// TIA Portal project "Homework-Traffic Light" (V16)

(* hardware
DEVICE "HMI_1"  KTP700 Basic PN
   slot 0: "HMI_1"  KTP700 Basic PN  6AV2 123-2GB03-0AX0  16.0.0.0
   slot 1: "HMI_RT_1"  KTP700 Basic PN  6AV2 123-2GB03-0AX0  16.0.0.0
   slot 5: "HMI_1.IE_CP_1"  PROFINET Interface  16.0.0.0
      slot 1: "PROFINET Interface_1"  PROFINET Interface
         slot 1: "Port_1"  Port
DEVICE "PC-System_1"  SIMATIC PC station
   slot 0: "SIMATIC PC station"  Rail  SIMATIC PC-Station  V1.0
      slot 125: "Stationmanager"  Station_Manager  V6.0.4
   slot 1: "HMI_RT_2"  WinCC RT Advanced  6AV2 104-0xxxx-xxxx  16.0.0.0
      slot 33792: "Computer interface"  Host interface
   slot 2: "IE general_1"  IE General  IE_CP  V8.2.0
DEVICE "PC-System_2"  SIMATIC PC station
   slot 0: "SIMATIC PC station"  Rail  SIMATIC PC-Station  V1.0
      slot 125: "Stationmanager"  Station_Manager  V6.0.4
   slot 1: "HMI_RT_3"  WinCC RT Professional  6AV2 105-0xxxx-xxxx  16.0.0.0
   slot 2: "IE general_1"  IE General  IE_CP  V8.2.0
DEVICE "S71500/ET200MP station_1"  S7-1500 station
   slot 0: "Rail_0"  Rack  6ES7 590-1***0-0AA0
   slot 1: "PLC_2"  CPU 1512C-1 PN  6ES7 512-1CK00-0AB0  V2.5
      slot 3: "CPU display_1"  6ES7591-1AA00-0AA0
      slot 32768: "PROFINET interface_1"  X1
   slot 2: "CM PtP RS232 HF_1"  CM PtP RS232 HF  6ES7 541-1AD00-0AB0  V1.0
   slot 3: "CM PtP RS232 HF_2"  CM PtP RS232 HF  6ES7 541-1AD00-0AB0  V1.0
*)

// ===== PLC "PLC_2"  CPU 1512C-1 PN =====

VAR_GLOBAL   // PLC tag table "Default tag table"
   "System_Byte" AT %MB7 : Byte;
   "FirstScan" AT %M7.0 : Bool;
   "DiagStatusUpdate" AT %M7.1 : Bool;
   "AlwaysTRUE" AT %M7.2 : Bool;
   "AlwaysFALSE" AT %M7.3 : Bool;
   "Clock_Byte" AT %MB8 : Byte;
   "Clock_10Hz" AT %M8.0 : Bool;
   "Clock_5Hz" AT %M8.1 : Bool;
   "Clock_2.5Hz" AT %M8.2 : Bool;
   "Clock_2Hz" AT %M8.3 : Bool;
   "Clock_1.25Hz" AT %M8.4 : Bool;
   "Clock_1Hz" AT %M8.5 : Bool;
   "Clock_0.625Hz" AT %M8.6 : Bool;
   "Clock_0.5Hz" AT %M8.7 : Bool;
   "Pulse1" AT %M0.0 : Bool;
   "Pulse2" AT %M0.1 : Bool;
   "Pulse3" AT %M0.2 : Bool;
   "Pulse4" AT %M0.3 : Bool;
   "Pulse5" AT %M0.4 : Bool;
   "Pulse6" AT %M0.5 : Bool;
   "Pulse_1s" AT %M0.6 : Bool;
   "Pulse7" AT %M0.7 : Bool;
   "Remain3" AT %M1.0 : Bool;
   "Remain1" AT %M1.1 : Bool;
   "Remain2" AT %M1.2 : Bool;
   "Remain4" AT %M1.3 : Bool;
   "Green_A" AT %Q4.0 : Bool;
   "Yellow_A" AT %Q4.1 : Bool;
   "Red_A" AT %Q4.2 : Bool;
   "Green_B" AT %Q4.3 : Bool;
   "Yellow_B" AT %Q4.4 : Bool;
   "Red_B" AT %Q4.5 : Bool;
   "Stop_System(1)" AT %I10.0 : Bool;
   "Start_System" AT %I10.1 : Bool;
   "Cross_Over" AT %M5.0 : Bool;
END_VAR

DATA_BLOCK "System Data"   // DB1
{ S7_Optimized_Access := 'TRUE' }
VERSION : 0.1
   VAR
      "Green A" : Bool;
      "Green B" : Bool;
      "Yellow A" : Bool;
      "Yellow B" : Bool;
      "Red A" : Bool;
      "Red B" : Bool;
      HMI_Update : Bool;
      Enable_PP1 : Bool;
      Enalbe_PP2 : Bool;
      Enalbe_PP3 : Bool;
      Start : Bool;
      Stop : Bool;
      RUN_System : Bool;
      HMI_SET : Bool;
      "Green A _Value" : DInt;
      "Green B_Value" : DInt;
      "Yellow A_value" : DInt;
      "Yellow B_value" : DInt;
      Red_A_value : DInt;
      Red_B_Value : DInt;
      HMI_Green_A : DInt;
      HMI_Green_B : DInt;
      HMI_Yellow_A : DInt;
      HMI_Yellow_B : DInt;
      HMI_Red_A : DInt;
      HMI_Red_B : DInt;
      Reset : Bool;
      Last_signal : Bool;
      Read_Time : DTL;
      RET_Val : Word;
      Time_day : Bool;
      Time_night : Bool;
      Visible_1 : Bool;
      Visible_2 : Bool;
      Mode : DInt;
      Cross : Bool;
   END_VAR
BEGIN
END_DATA_BLOCK

DATA_BLOCK "7SEG_Convert1"   // DB6
{ S7_Optimized_Access := 'TRUE' }
VERSION : 0.1
// stored: InstanceOfName Convert_BCD_7SEG
"Convert_BCD_7SEG"
BEGIN
END_DATA_BLOCK

DATA_BLOCK "Data"   // DB8
{ S7_Optimized_Access := 'TRUE' }
VERSION : 0.1
   VAR
      HMI_Cancel : Bool;
      "Green A _Value" : DInt;
      "Green B_Value" : DInt;
      "1Timer_TImerA" : DInt;
      "1Timer_TimerB" : DInt;
      "4Timer_Timer" : DInt;
      Counter_Time : DInt;
      Time_Max_Counter : DInt;
      "Yellow A_Value" : DInt;
      "Yellow B_Value" : DInt;
      "Red A_Value" : DInt;
      "Red B_Value" : DInt;
      GY_Value_A : DInt;
      GY_Value_B : DInt;
      "1Timer_Remain_LightB" : DInt;
      "1Timer_Remain_LightA" : DInt;
      TIme_LIGHT_A : DInt;
      Time_LIGHT_B : DInt;
      Timer_Light_YellowB_Remain : DInt;
      Timer_Light_YellowA_Remain : DInt;
      Counter_remain_Light_A : DInt;
      Counter_remain_Light_B : DInt;
      DEC_DIV_A : Int;
      DEC_DIV_B : Int;
      DEC_MOD_A : Int;
      DEC_MOD_B : Int;
      Remain_DEC_A : Int;
      Remain_DEC_B : Int;
      "7SEG_DIV_A" : Byte;
      "7SEG_MOD_A" : Byte;
      "7SEG_DIV_B" : Byte;
      "7SEG_MOD_B" : Byte;
      Cross_Remain : DInt;
   END_VAR
BEGIN
END_DATA_BLOCK

DATA_BLOCK "7SEG_Convert2"   // DB9
{ S7_Optimized_Access := 'TRUE' }
VERSION : 0.1
// stored: InstanceOfName Convert_BCD_7SEG
"Convert_BCD_7SEG"
BEGIN
END_DATA_BLOCK

DATA_BLOCK "7SEG_Convert3"   // DB10
{ S7_Optimized_Access := 'TRUE' }
VERSION : 0.1
// stored: InstanceOfName Convert_BCD_7SEG
"Convert_BCD_7SEG"
BEGIN
END_DATA_BLOCK

DATA_BLOCK "7SEG_Convert4"   // DB11
{ S7_Optimized_Access := 'TRUE' }
VERSION : 0.1
// stored: InstanceOfName Convert_BCD_7SEG
"Convert_BCD_7SEG"
BEGIN
END_DATA_BLOCK

// folder: System blocks/Program resources

DATA_BLOCK "Timer1"   // DB2
{ S7_Optimized_Access := 'TRUE' }
AUTHOR : Simatic
FAMILY : IEC
NAME : IEC_TMR
VERSION : 1.0
// stored: InstanceOfName IEC_TIMER
"IEC_TIMER"
BEGIN
END_DATA_BLOCK

DATA_BLOCK "Timer2"   // DB3
{ S7_Optimized_Access := 'TRUE' }
AUTHOR : Simatic
FAMILY : IEC
NAME : IEC_TMR
VERSION : 1.0
// stored: InstanceOfName IEC_TIMER
"IEC_TIMER"
BEGIN
END_DATA_BLOCK

DATA_BLOCK "Timer3"   // DB4
{ S7_Optimized_Access := 'TRUE' }
AUTHOR : Simatic
FAMILY : IEC
NAME : IEC_TMR
VERSION : 1.0
// stored: InstanceOfName IEC_TIMER
"IEC_TIMER"
BEGIN
END_DATA_BLOCK

DATA_BLOCK "Timer4"   // DB5
{ S7_Optimized_Access := 'TRUE' }
AUTHOR : Simatic
FAMILY : IEC
NAME : IEC_TMR
VERSION : 1.0
// stored: InstanceOfName IEC_TIMER
"IEC_TIMER"
BEGIN
END_DATA_BLOCK

DATA_BLOCK "T1"   // DB7
{ S7_Optimized_Access := 'TRUE' }
AUTHOR : Simatic
FAMILY : IEC
NAME : IEC_TMR
VERSION : 1.0
// stored: InstanceOfName IEC_TIMER
"IEC_TIMER"
BEGIN
END_DATA_BLOCK

DATA_BLOCK "T2"   // DB13
{ S7_Optimized_Access := 'TRUE' }
AUTHOR : Simatic
FAMILY : IEC
NAME : IEC_TMR
VERSION : 1.0
// stored: InstanceOfName IEC_TIMER
"IEC_TIMER"
BEGIN
END_DATA_BLOCK

// folder: (top level)

FUNCTION_BLOCK "Convert_BCD_7SEG"   // FB1, SCL
{ S7_Optimized_Access := 'TRUE' }
VERSION : 0.1
   VAR_INPUT
      BCD_Val : Int;
   END_VAR
   VAR_OUTPUT
      "7SEG_Val" : Byte;
   END_VAR
   VAR_TEMP
      tmp : Byte;
   END_VAR
BEGIN
   #tmp := 0;
   IF #BCD_Val =0 THEN
       #tmp := 63;
   END_IF;
   IF #BCD_Val = 1 THEN
       #tmp := 6;
   END_IF;
   IF #BCD_Val = 2 THEN
       #tmp := 91;
   END_IF;
   IF #BCD_Val = 3 THEN
       #tmp := 79;
   END_IF;
   IF #BCD_Val = 4 THEN
       #tmp := 102;
   END_IF;
   IF #BCD_Val = 5 THEN
       #tmp := 109;
   END_IF;
   IF #BCD_Val = 6 THEN
       #tmp := 125;
   END_IF;
   IF #BCD_Val = 7 THEN
       #tmp := 7;
   END_IF;
   IF #BCD_Val = 8 THEN
       #tmp := 127;
   END_IF;
   IF #BCD_Val = 9 THEN
       #tmp := 111;
   END_IF;
   #"7SEG_Val" := #tmp;
END_FUNCTION_BLOCK

FUNCTION "PP2_4Timer" : Void   // FC1, LAD
{ S7_Optimized_Access := 'TRUE' }
VERSION : 0.1
   VAR_TEMP   // added for the SCL form of the ladder/FBD networks
      _w1 : Bool;
   END_VAR
BEGIN

REGION Network 1
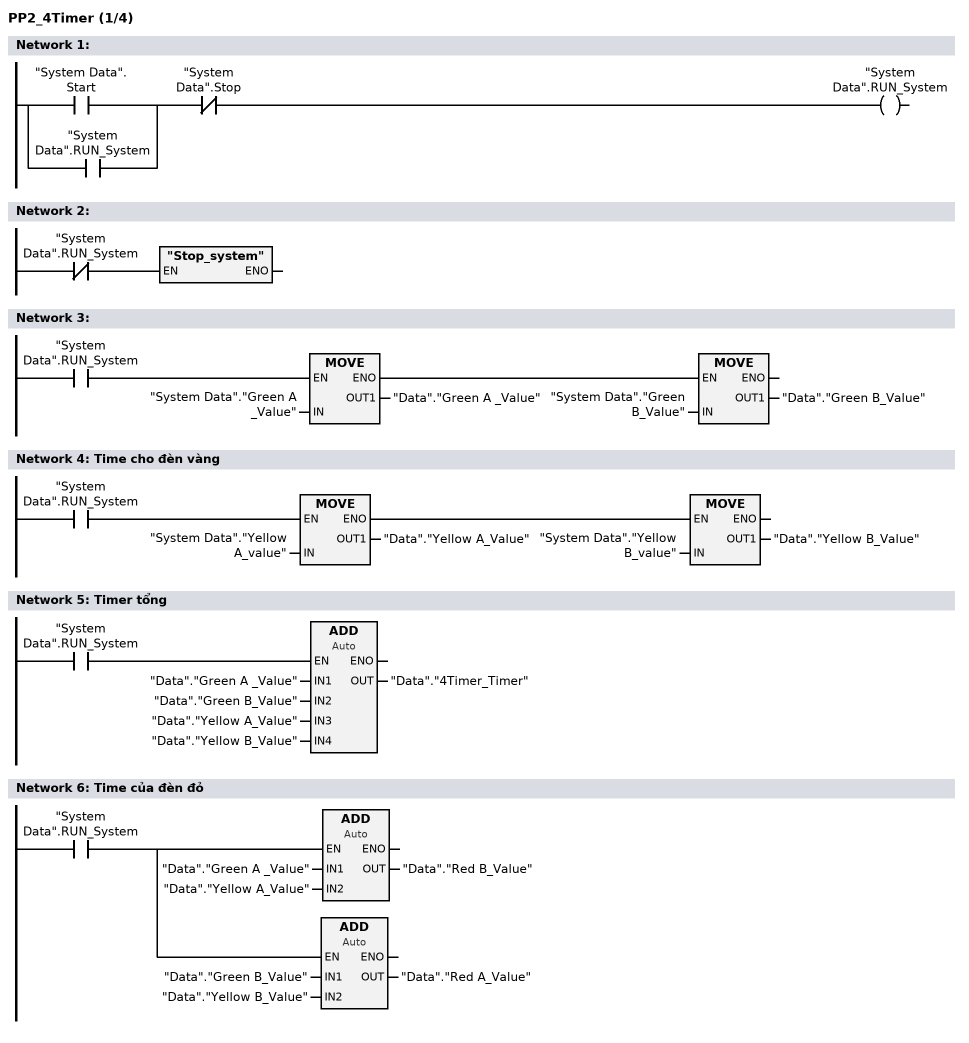
   RUNG wire#powerrail
      Contact( "System Data".Start )
      wire#w1
      I_Contact( "System Data".Stop )
      Coil( "System Data".RUN_System )
   END_RUNG
   RUNG wire#powerrail
      Contact( "System Data".RUN_System )
   END_RUNG wire#w1
   // the same network as SCL:
   "System Data".RUN_System := ("System Data".Start OR "System Data".RUN_System) AND NOT "System Data".Stop;
END_REGION

REGION Network 2
   RUNG wire#powerrail
      I_Contact( "System Data".RUN_System )
      "Stop_system"()
   END_RUNG
   // the same network as SCL:
   IF NOT "System Data".RUN_System THEN "Stop_system"(); END_IF;
END_REGION

REGION Network 3
   RUNG wire#powerrail
      Contact( "System Data".RUN_System )
      Move(in := "System Data"."Green A _Value", out1 => "Data"."Green A _Value")
      Move(in := "System Data"."Green B_Value", out1 => "Data"."Green B_Value")
   END_RUNG
   // the same network as SCL:
   IF "System Data".RUN_System THEN
       "Data"."Green A _Value" := "System Data"."Green A _Value";
       "Data"."Green B_Value" := "System Data"."Green B_Value";
   END_IF;
END_REGION

REGION Network 4: Time cho đèn vàng
   RUNG wire#powerrail
      Contact( "System Data".RUN_System )
      Move(in := "System Data"."Yellow A_value", out1 => "Data"."Yellow A_Value")
      Move(in := "System Data"."Yellow B_value", out1 => "Data"."Yellow B_Value")
   END_RUNG
   // the same network as SCL:
   IF "System Data".RUN_System THEN
       "Data"."Yellow A_Value" := "System Data"."Yellow A_value";
       "Data"."Yellow B_Value" := "System Data"."Yellow B_value";
   END_IF;
END_REGION

REGION Network 5: Timer tổng
   RUNG wire#powerrail
      Contact( "System Data".RUN_System )
      Add(in1 := "Data"."Green A _Value", in2 := "Data"."Green B_Value", in3 := "Data"."Yellow A_Value", in4 := "Data"."Yellow B_Value", out => "Data"."4Timer_Timer")
   END_RUNG
   // the same network as SCL:
   IF "System Data".RUN_System THEN
       "Data"."4Timer_Timer" := "Data"."Green A _Value" + "Data"."Green B_Value" + "Data"."Yellow A_Value" + "Data"."Yellow B_Value";
   END_IF;
END_REGION

REGION Network 6: Time của đèn đỏ
   RUNG wire#powerrail
      Contact( "System Data".RUN_System )
      wire#w1
      Add(in1 := "Data"."Green A _Value", in2 := "Data"."Yellow A_Value", out => "Data"."Red B_Value")
   END_RUNG
   RUNG wire#w1
      Add(in1 := "Data"."Green B_Value", in2 := "Data"."Yellow B_Value", out => "Data"."Red A_Value")
   END_RUNG
   // the same network as SCL:
   IF "System Data".RUN_System THEN
       "Data"."Red B_Value" := "Data"."Green A _Value" + "Data"."Yellow A_Value";
       "Data"."Red A_Value" := "Data"."Green B_Value" + "Data"."Yellow B_Value";
   END_IF;
END_REGION

REGION Network 7
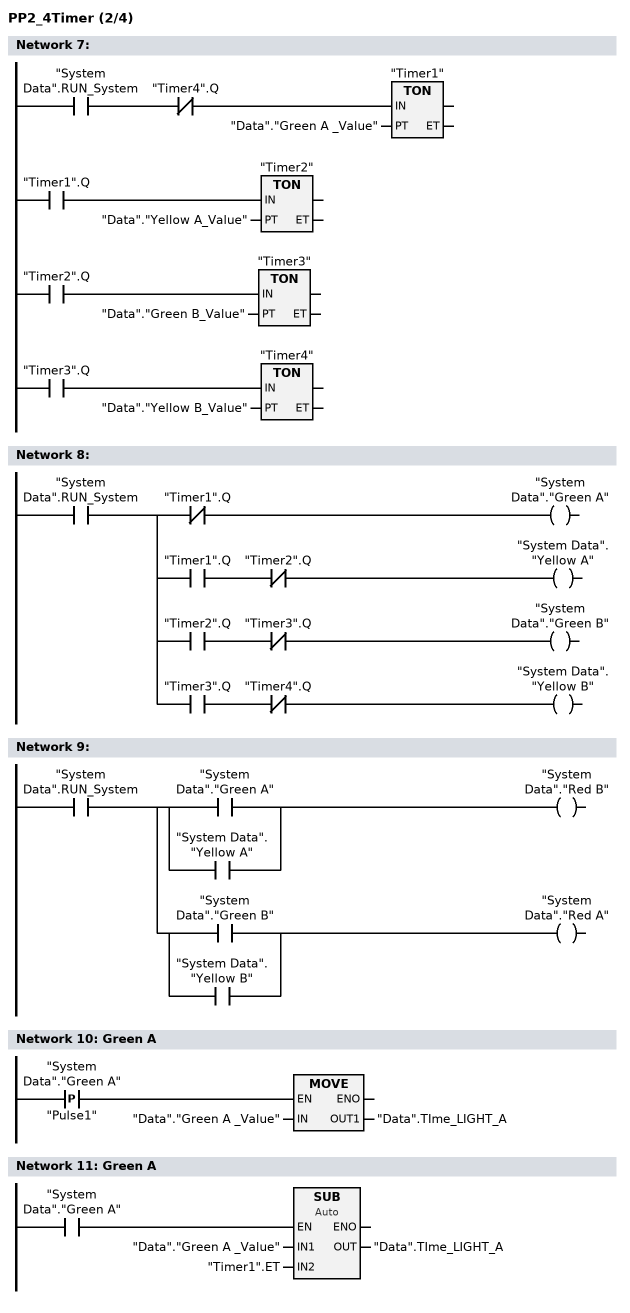
   "Timer1".TON(IN := "System Data".RUN_System AND NOT "Timer4".Q, PT := "Data"."Green A _Value");
   "Timer2".TON(IN := "Timer1".Q, PT := "Data"."Yellow A_Value");
   "Timer3".TON(IN := "Timer2".Q, PT := "Data"."Green B_Value");
   "Timer4".TON(IN := "Timer3".Q, PT := "Data"."Yellow B_Value");
END_REGION

REGION Network 8
   RUNG wire#powerrail
      Contact( "System Data".RUN_System )
      wire#w1
      I_Contact( "Timer1".Q )
      Coil( "System Data"."Green A" )
   END_RUNG
   RUNG wire#w1
      Contact( "Timer1".Q )
      I_Contact( "Timer2".Q )
      Coil( "System Data"."Yellow A" )
   END_RUNG
   RUNG wire#w1
      Contact( "Timer2".Q )
      I_Contact( "Timer3".Q )
      Coil( "System Data"."Green B" )
   END_RUNG
   RUNG wire#w1
      Contact( "Timer3".Q )
      I_Contact( "Timer4".Q )
      Coil( "System Data"."Yellow B" )
   END_RUNG
   // the same network as SCL:
   "System Data"."Green A" := "System Data".RUN_System AND NOT "Timer1".Q;
   "System Data"."Yellow A" := "System Data".RUN_System AND "Timer1".Q AND NOT "Timer2".Q;
   "System Data"."Green B" := "System Data".RUN_System AND "Timer2".Q AND NOT "Timer3".Q;
   "System Data"."Yellow B" := "System Data".RUN_System AND "Timer3".Q AND NOT "Timer4".Q;
END_REGION

REGION Network 9
   RUNG wire#powerrail
      Contact( "System Data".RUN_System )
      wire#w1
      Contact( "System Data"."Green A" )
      wire#w2
      Coil( "System Data"."Red B" )
   END_RUNG
   RUNG wire#w1
      Contact( "System Data"."Yellow A" )
   END_RUNG wire#w2
   RUNG wire#w1
      Contact( "System Data"."Green B" )
      wire#w3
      Coil( "System Data"."Red A" )
   END_RUNG
   RUNG wire#w1
      Contact( "System Data"."Yellow B" )
   END_RUNG wire#w3
   // the same network as SCL:
   "System Data"."Red B" := "System Data".RUN_System AND ("System Data"."Green A" OR "System Data"."Yellow A");
   "System Data"."Red A" := "System Data".RUN_System AND ("System Data"."Green B" OR "System Data"."Yellow B");
END_REGION

REGION Network 10: Green A
   RUNG wire#powerrail
      P_Contact(operand := "System Data"."Green A", bit := "Pulse1")
      Move(in := "Data"."Green A _Value", out1 => "Data".TIme_LIGHT_A)
   END_RUNG
   // the same network as SCL:
   #_w1 := "System Data"."Green A" AND NOT "Pulse1";   // rising edge of "System Data"."Green A"
   "Pulse1" := "System Data"."Green A";
   IF #_w1 THEN "Data".TIme_LIGHT_A := "Data"."Green A _Value"; END_IF;
END_REGION

REGION Network 11: Green A
   RUNG wire#powerrail
      Contact( "System Data"."Green A" )
      Sub(in1 := "Data"."Green A _Value", in2 := "Timer1".ET, out => "Data".TIme_LIGHT_A)
   END_RUNG
   // the same network as SCL:
   IF "System Data"."Green A" THEN "Data".TIme_LIGHT_A := "Data"."Green A _Value" - "Timer1".ET; END_IF;
END_REGION

REGION Network 12: Yellow A
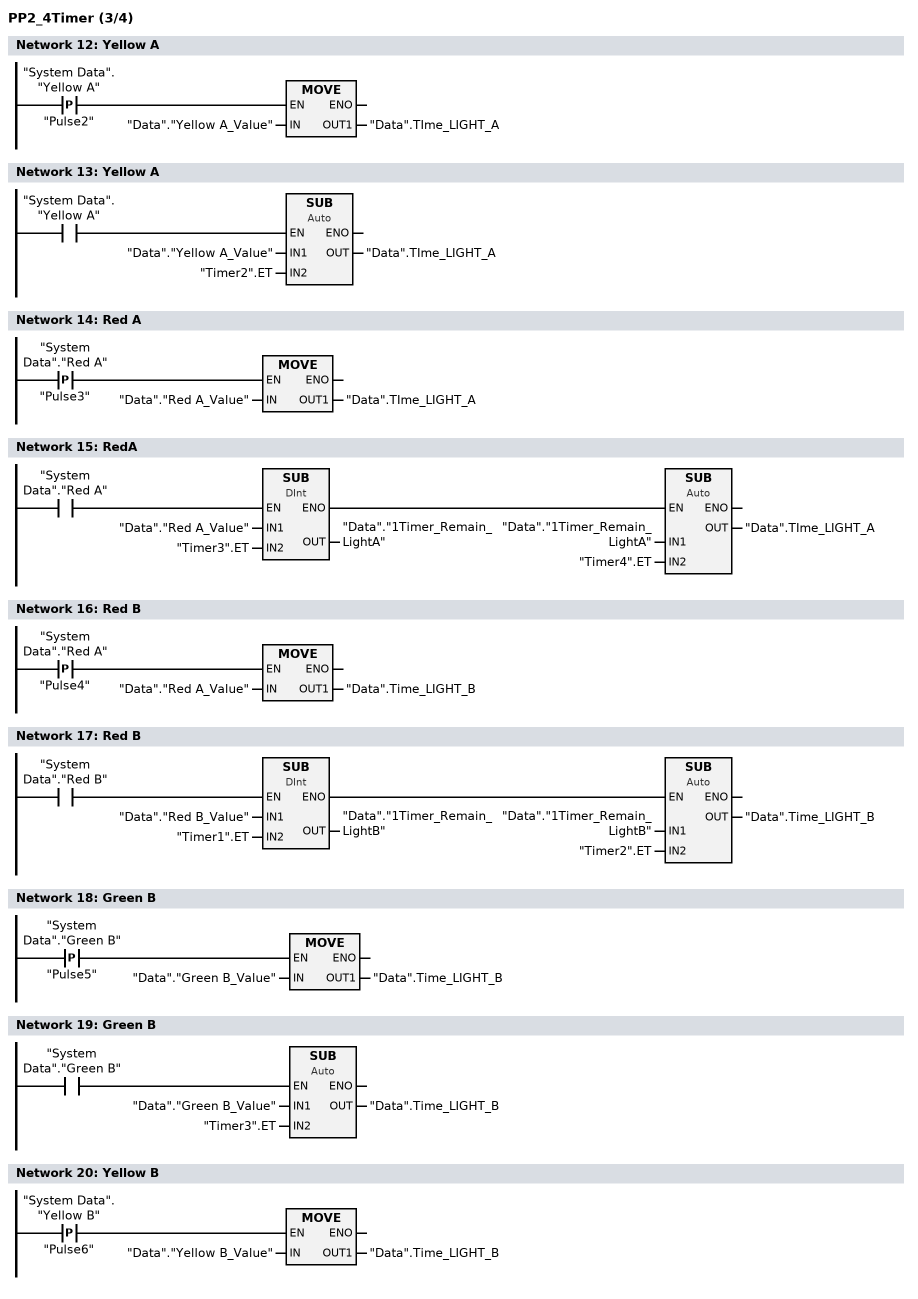
   RUNG wire#powerrail
      P_Contact(operand := "System Data"."Yellow A", bit := "Pulse2")
      Move(in := "Data"."Yellow A_Value", out1 => "Data".TIme_LIGHT_A)
   END_RUNG
   // the same network as SCL:
   #_w1 := "System Data"."Yellow A" AND NOT "Pulse2";   // rising edge of "System Data"."Yellow A"
   "Pulse2" := "System Data"."Yellow A";
   IF #_w1 THEN "Data".TIme_LIGHT_A := "Data"."Yellow A_Value"; END_IF;
END_REGION

REGION Network 13: Yellow A
   RUNG wire#powerrail
      Contact( "System Data"."Yellow A" )
      Sub(in1 := "Data"."Yellow A_Value", in2 := "Timer2".ET, out => "Data".TIme_LIGHT_A)
   END_RUNG
   // the same network as SCL:
   IF "System Data"."Yellow A" THEN "Data".TIme_LIGHT_A := "Data"."Yellow A_Value" - "Timer2".ET; END_IF;
END_REGION

REGION Network 14: Red A
   RUNG wire#powerrail
      P_Contact(operand := "System Data"."Red A", bit := "Pulse3")
      Move(in := "Data"."Red A_Value", out1 => "Data".TIme_LIGHT_A)
   END_RUNG
   // the same network as SCL:
   #_w1 := "System Data"."Red A" AND NOT "Pulse3";   // rising edge of "System Data"."Red A"
   "Pulse3" := "System Data"."Red A";
   IF #_w1 THEN "Data".TIme_LIGHT_A := "Data"."Red A_Value"; END_IF;
END_REGION

REGION Network 15: RedA
   RUNG wire#powerrail
      Contact( "System Data"."Red A" )
      { S7_Templates := "SrcType := DInt" } Sub(in1 := "Data"."Red A_Value", in2 := "Timer3".ET, out => "Data"."1Timer_Remain_LightA")
      Sub(in1 := "Data"."1Timer_Remain_LightA", in2 := "Timer4".ET, out => "Data".TIme_LIGHT_A)
   END_RUNG
   // the same network as SCL:
   IF "System Data"."Red A" THEN
       "Data"."1Timer_Remain_LightA" := "Data"."Red A_Value" - "Timer3".ET;
       "Data".TIme_LIGHT_A := "Data"."1Timer_Remain_LightA" - "Timer4".ET;
   END_IF;
END_REGION

REGION Network 16: Red B
   RUNG wire#powerrail
      P_Contact(operand := "System Data"."Red A", bit := "Pulse4")
      Move(in := "Data"."Red A_Value", out1 => "Data".Time_LIGHT_B)
   END_RUNG
   // the same network as SCL:
   #_w1 := "System Data"."Red A" AND NOT "Pulse4";   // rising edge of "System Data"."Red A"
   "Pulse4" := "System Data"."Red A";
   IF #_w1 THEN "Data".Time_LIGHT_B := "Data"."Red A_Value"; END_IF;
END_REGION

REGION Network 17: Red B
   RUNG wire#powerrail
      Contact( "System Data"."Red B" )
      { S7_Templates := "SrcType := DInt" } Sub(in1 := "Data"."Red B_Value", in2 := "Timer1".ET, out => "Data"."1Timer_Remain_LightB")
      Sub(in1 := "Data"."1Timer_Remain_LightB", in2 := "Timer2".ET, out => "Data".Time_LIGHT_B)
   END_RUNG
   // the same network as SCL:
   IF "System Data"."Red B" THEN
       "Data"."1Timer_Remain_LightB" := "Data"."Red B_Value" - "Timer1".ET;
       "Data".Time_LIGHT_B := "Data"."1Timer_Remain_LightB" - "Timer2".ET;
   END_IF;
END_REGION

REGION Network 18: Green B
   RUNG wire#powerrail
      P_Contact(operand := "System Data"."Green B", bit := "Pulse5")
      Move(in := "Data"."Green B_Value", out1 => "Data".Time_LIGHT_B)
   END_RUNG
   // the same network as SCL:
   #_w1 := "System Data"."Green B" AND NOT "Pulse5";   // rising edge of "System Data"."Green B"
   "Pulse5" := "System Data"."Green B";
   IF #_w1 THEN "Data".Time_LIGHT_B := "Data"."Green B_Value"; END_IF;
END_REGION

REGION Network 19: Green B
   RUNG wire#powerrail
      Contact( "System Data"."Green B" )
      Sub(in1 := "Data"."Green B_Value", in2 := "Timer3".ET, out => "Data".Time_LIGHT_B)
   END_RUNG
   // the same network as SCL:
   IF "System Data"."Green B" THEN "Data".Time_LIGHT_B := "Data"."Green B_Value" - "Timer3".ET; END_IF;
END_REGION

REGION Network 20: Yellow B
   RUNG wire#powerrail
      P_Contact(operand := "System Data"."Yellow B", bit := "Pulse6")
      Move(in := "Data"."Yellow B_Value", out1 => "Data".Time_LIGHT_B)
   END_RUNG
   // the same network as SCL:
   #_w1 := "System Data"."Yellow B" AND NOT "Pulse6";   // rising edge of "System Data"."Yellow B"
   "Pulse6" := "System Data"."Yellow B";
   IF #_w1 THEN "Data".Time_LIGHT_B := "Data"."Yellow B_Value"; END_IF;
END_REGION

REGION Network 21: Yellow B
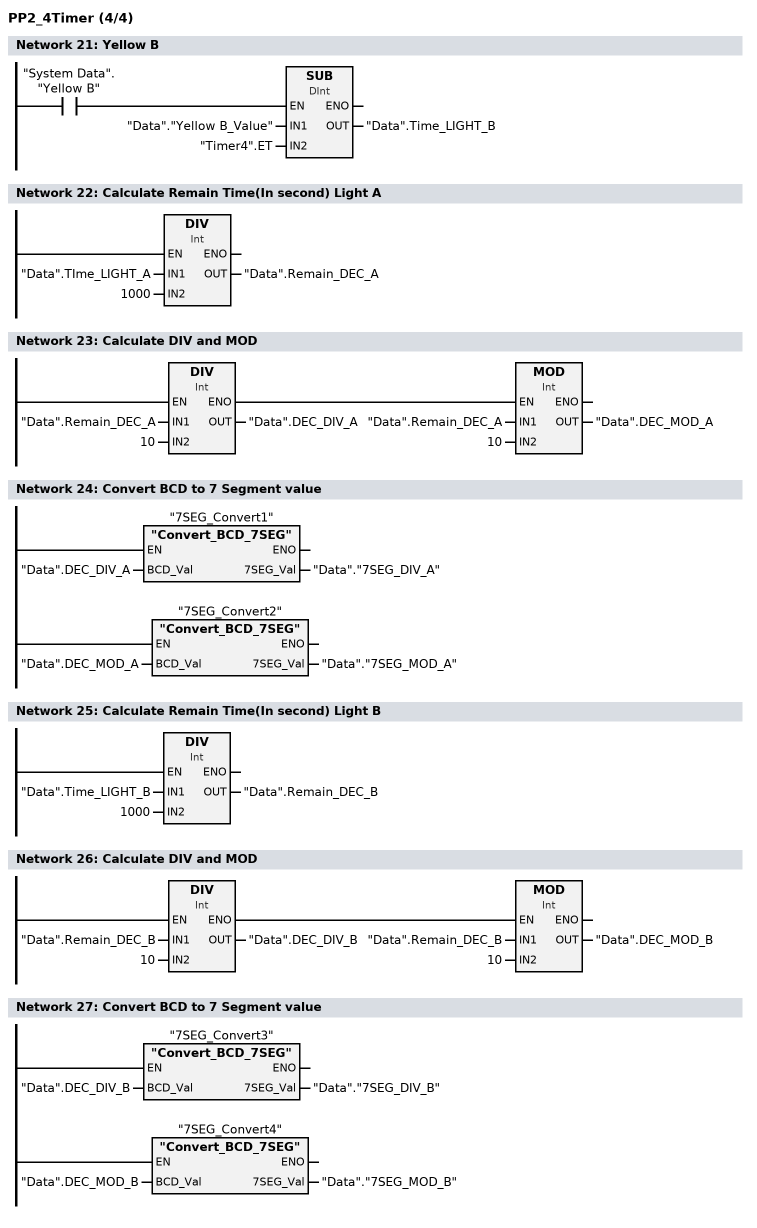
   RUNG wire#powerrail
      Contact( "System Data"."Yellow B" )
      { S7_Templates := "SrcType := DInt" } Sub(in1 := "Data"."Yellow B_Value", in2 := "Timer4".ET, out => "Data".Time_LIGHT_B)
   END_RUNG
   // the same network as SCL:
   IF "System Data"."Yellow B" THEN "Data".Time_LIGHT_B := "Data"."Yellow B_Value" - "Timer4".ET; END_IF;
END_REGION

REGION Network 22: Calculate Remain Time(In second) Light A
   RUNG wire#powerrail
      { S7_Templates := "SrcType := Int" } Div(in1 := "Data".TIme_LIGHT_A, in2 := 1000, out => "Data".Remain_DEC_A)
   END_RUNG
   // the same network as SCL:
   "Data".Remain_DEC_A := "Data".TIme_LIGHT_A / 1000;
END_REGION

REGION Network 23: Calculate DIV and MOD
   RUNG wire#powerrail
      { S7_Templates := "SrcType := Int" } Div(in1 := "Data".Remain_DEC_A, in2 := 10, out => "Data".DEC_DIV_A)
      { S7_Templates := "SrcType := Int" } Mod(in1 := "Data".Remain_DEC_A, in2 := 10, out => "Data".DEC_MOD_A)
   END_RUNG
   // the same network as SCL:
   "Data".DEC_DIV_A := "Data".Remain_DEC_A / 10;
   "Data".DEC_MOD_A := "Data".Remain_DEC_A MOD 10;
END_REGION

REGION Network 24: Convert BCD to 7 Segment value
   RUNG wire#powerrail
      "7SEG_Convert1"(BCD_Val := "Data".DEC_DIV_A, "7SEG_Val" => "Data"."7SEG_DIV_A")
   END_RUNG
   RUNG wire#powerrail
      "7SEG_Convert2"(BCD_Val := "Data".DEC_MOD_A, "7SEG_Val" => "Data"."7SEG_MOD_A")
   END_RUNG
   // the same network as SCL:
   "7SEG_Convert1"(BCD_Val := "Data".DEC_DIV_A, "7SEG_Val" => "Data"."7SEG_DIV_A");   // "Convert_BCD_7SEG"
   "7SEG_Convert2"(BCD_Val := "Data".DEC_MOD_A, "7SEG_Val" => "Data"."7SEG_MOD_A");   // "Convert_BCD_7SEG"
END_REGION

REGION Network 25: Calculate Remain Time(In second) Light B
   RUNG wire#powerrail
      { S7_Templates := "SrcType := Int" } Div(in1 := "Data".Time_LIGHT_B, in2 := 1000, out => "Data".Remain_DEC_B)
   END_RUNG
   // the same network as SCL:
   "Data".Remain_DEC_B := "Data".Time_LIGHT_B / 1000;
END_REGION

REGION Network 26: Calculate DIV and MOD
   RUNG wire#powerrail
      { S7_Templates := "SrcType := Int" } Div(in1 := "Data".Remain_DEC_B, in2 := 10, out => "Data".DEC_DIV_B)
      { S7_Templates := "SrcType := Int" } Mod(in1 := "Data".Remain_DEC_B, in2 := 10, out => "Data".DEC_MOD_B)
   END_RUNG
   // the same network as SCL:
   "Data".DEC_DIV_B := "Data".Remain_DEC_B / 10;
   "Data".DEC_MOD_B := "Data".Remain_DEC_B MOD 10;
END_REGION

REGION Network 27: Convert BCD to 7 Segment value
   RUNG wire#powerrail
      "7SEG_Convert3"(BCD_Val := "Data".DEC_DIV_B, "7SEG_Val" => "Data"."7SEG_DIV_B")
   END_RUNG
   RUNG wire#powerrail
      "7SEG_Convert4"(BCD_Val := "Data".DEC_MOD_B, "7SEG_Val" => "Data"."7SEG_MOD_B")
   END_RUNG
   // the same network as SCL:
   "7SEG_Convert3"(BCD_Val := "Data".DEC_DIV_B, "7SEG_Val" => "Data"."7SEG_DIV_B");   // "Convert_BCD_7SEG"
   "7SEG_Convert4"(BCD_Val := "Data".DEC_MOD_B, "7SEG_Val" => "Data"."7SEG_MOD_B");   // "Convert_BCD_7SEG"
END_REGION
END_FUNCTION

FUNCTION "PP1_1Timer" : Void   // FC2, LAD
{ S7_Optimized_Access := 'TRUE' }
VERSION : 0.1
   VAR_TEMP   // added for the SCL form of the ladder/FBD networks
      _w1 : Bool;
   END_VAR
BEGIN

REGION Network 1
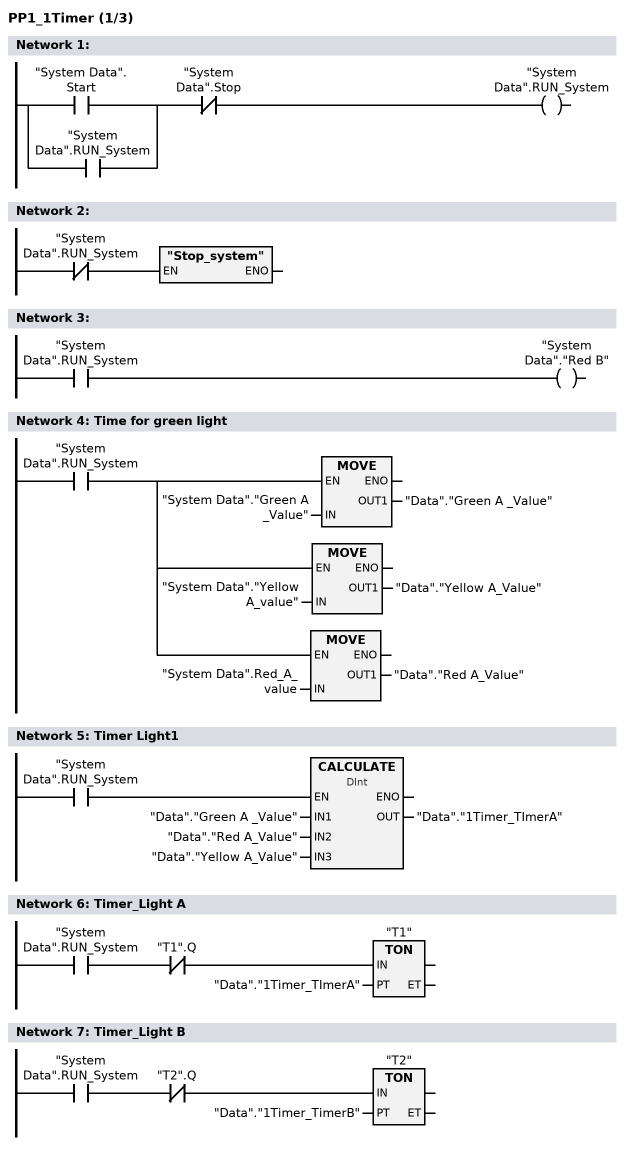
   RUNG wire#powerrail
      Contact( "System Data".Start )
      wire#w1
      I_Contact( "System Data".Stop )
      Coil( "System Data".RUN_System )
   END_RUNG
   RUNG wire#powerrail
      Contact( "System Data".RUN_System )
   END_RUNG wire#w1
   // the same network as SCL:
   "System Data".RUN_System := ("System Data".Start OR "System Data".RUN_System) AND NOT "System Data".Stop;
END_REGION

REGION Network 2
   RUNG wire#powerrail
      I_Contact( "System Data".RUN_System )
      "Stop_system"()
   END_RUNG
   // the same network as SCL:
   IF NOT "System Data".RUN_System THEN "Stop_system"(); END_IF;
END_REGION

REGION Network 3
   RUNG wire#powerrail
      Contact( "System Data".RUN_System )
      Coil( "System Data"."Red B" )
   END_RUNG
   // the same network as SCL:
   "System Data"."Red B" := "System Data".RUN_System;
END_REGION

REGION Network 4: Time for green light
   RUNG wire#powerrail
      Contact( "System Data".RUN_System )
      wire#w1
      Move(in := "System Data"."Green A _Value", out1 => "Data"."Green A _Value")
   END_RUNG
   RUNG wire#w1
      Move(in := "System Data"."Yellow A_value", out1 => "Data"."Yellow A_Value")
   END_RUNG
   RUNG wire#w1
      Move(in := "System Data".Red_A_value, out1 => "Data"."Red A_Value")
   END_RUNG
   // the same network as SCL:
   IF "System Data".RUN_System THEN
       "Data"."Green A _Value" := "System Data"."Green A _Value";
       "Data"."Yellow A_Value" := "System Data"."Yellow A_value";
       "Data"."Red A_Value" := "System Data".Red_A_value;
   END_IF;
END_REGION

REGION Network 5: Timer Light1
   RUNG wire#powerrail
      Contact( "System Data".RUN_System )
      { S7_Templates := "SrcType := DInt"; S7_Expression := "IN1+IN2+IN3" } Calculate(in1 := "Data"."Green A _Value", in2 := "Data"."Red A_Value", in3 := "Data"."Yellow A_Value", out => "Data"."1Timer_TImerA")
   END_RUNG
   // the same network as SCL:
   IF "System Data".RUN_System THEN
       "Data"."1Timer_TImerA" := "Data"."Green A _Value"+"Data"."Red A_Value"+"Data"."Yellow A_Value";
   END_IF;
END_REGION

REGION Network 6: Timer_Light A
   "T1".TON(IN := "System Data".RUN_System AND NOT "T1".Q, PT := "Data"."1Timer_TImerA");
END_REGION

REGION Network 7: Timer_Light B
   "T2".TON(IN := "System Data".RUN_System AND NOT "T2".Q, PT := "Data"."1Timer_TimerB");
END_REGION

REGION Network 8: Light A
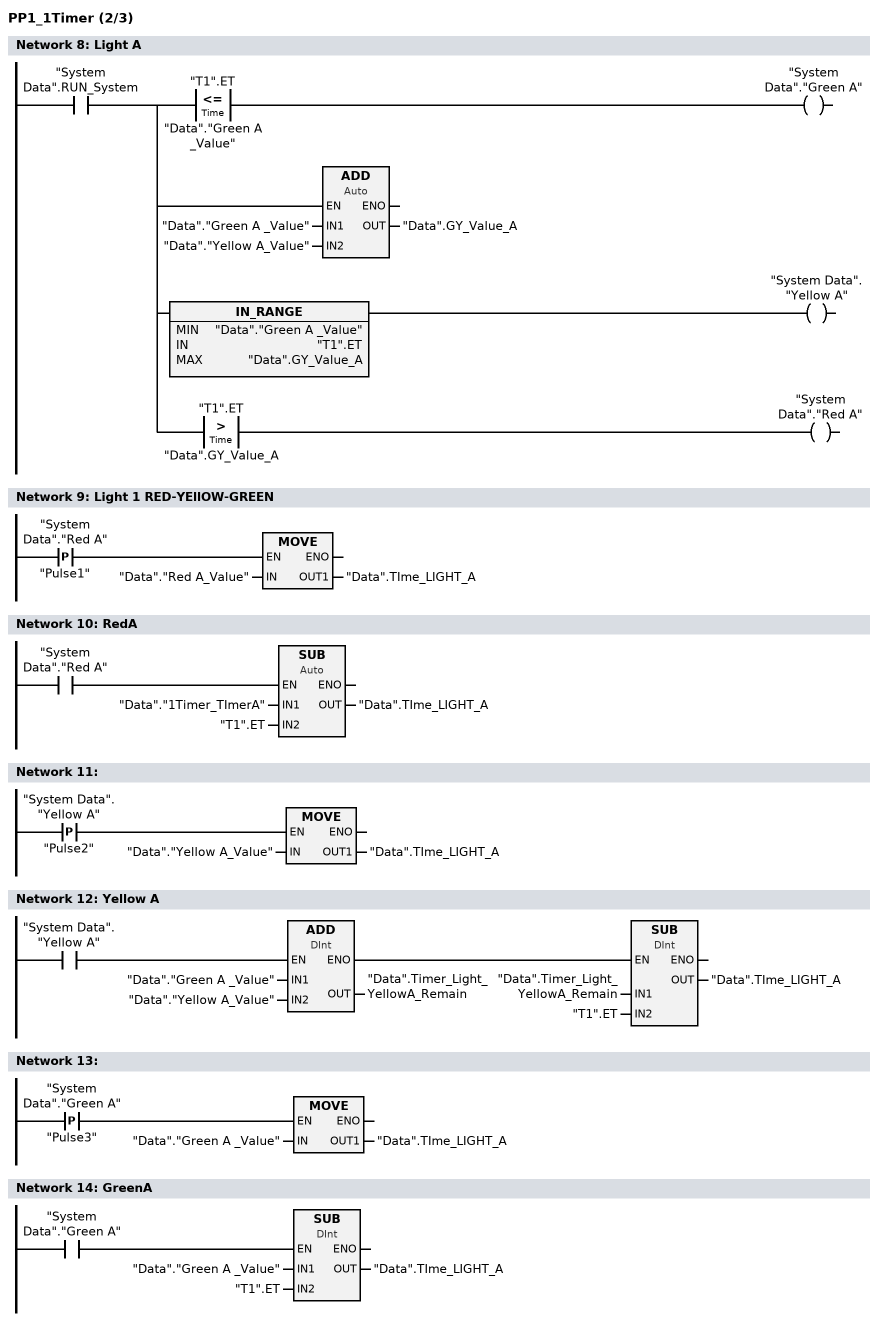
   RUNG wire#powerrail
      Contact( "System Data".RUN_System )
      wire#w1
      { S7_Templates := "SrcType := Time" } LE_Contact(in1 := "T1".ET, in2 := "Data"."Green A _Value")
      Coil( "System Data"."Green A" )
   END_RUNG
   RUNG wire#w1
      Add(in1 := "Data"."Green A _Value", in2 := "Data"."Yellow A_Value", out => "Data".GY_Value_A)
   END_RUNG
   RUNG wire#w1
      { S7_Templates := "SrcType := DInt" } InRange(min := "Data"."Green A _Value", in := "T1".ET, max := "Data".GY_Value_A)
      Coil( "System Data"."Yellow A" )
   END_RUNG
   RUNG wire#w1
      { S7_Templates := "SrcType := Time" } GT_Contact(in1 := "T1".ET, in2 := "Data".GY_Value_A)
      Coil( "System Data"."Red A" )
   END_RUNG
   // the same network as SCL:
   "System Data"."Green A" := "System Data".RUN_System AND ("T1".ET <= "Data"."Green A _Value");
   IF "System Data".RUN_System THEN
       "Data".GY_Value_A := "Data"."Green A _Value" + "Data"."Yellow A_Value";
   END_IF;
   "System Data"."Yellow A" := "System Data".RUN_System AND ("Data"."Green A _Value" <= "T1".ET) AND ("T1".ET <= "Data".GY_Value_A);
   "System Data"."Red A" := "System Data".RUN_System AND ("T1".ET > "Data".GY_Value_A);
END_REGION

REGION Network 9: Light 1 RED-YEllOW-GREEN
   RUNG wire#powerrail
      P_Contact(operand := "System Data"."Red A", bit := "Pulse1")
      Move(in := "Data"."Red A_Value", out1 => "Data".TIme_LIGHT_A)
   END_RUNG
   // the same network as SCL:
   #_w1 := "System Data"."Red A" AND NOT "Pulse1";   // rising edge of "System Data"."Red A"
   "Pulse1" := "System Data"."Red A";
   IF #_w1 THEN "Data".TIme_LIGHT_A := "Data"."Red A_Value"; END_IF;
END_REGION

REGION Network 10: RedA
   RUNG wire#powerrail
      Contact( "System Data"."Red A" )
      Sub(in1 := "Data"."1Timer_TImerA", in2 := "T1".ET, out => "Data".TIme_LIGHT_A)
   END_RUNG
   // the same network as SCL:
   IF "System Data"."Red A" THEN "Data".TIme_LIGHT_A := "Data"."1Timer_TImerA" - "T1".ET; END_IF;
END_REGION

REGION Network 11
   RUNG wire#powerrail
      P_Contact(operand := "System Data"."Yellow A", bit := "Pulse2")
      Move(in := "Data"."Yellow A_Value", out1 => "Data".TIme_LIGHT_A)
   END_RUNG
   // the same network as SCL:
   #_w1 := "System Data"."Yellow A" AND NOT "Pulse2";   // rising edge of "System Data"."Yellow A"
   "Pulse2" := "System Data"."Yellow A";
   IF #_w1 THEN "Data".TIme_LIGHT_A := "Data"."Yellow A_Value"; END_IF;
END_REGION

REGION Network 12: Yellow A
   RUNG wire#powerrail
      Contact( "System Data"."Yellow A" )
      { S7_Templates := "SrcType := DInt" } Add(in1 := "Data"."Green A _Value", in2 := "Data"."Yellow A_Value", out => "Data".Timer_Light_YellowA_Remain)
      { S7_Templates := "SrcType := DInt" } Sub(in1 := "Data".Timer_Light_YellowA_Remain, in2 := "T1".ET, out => "Data".TIme_LIGHT_A)
   END_RUNG
   // the same network as SCL:
   IF "System Data"."Yellow A" THEN
       "Data".Timer_Light_YellowA_Remain := "Data"."Green A _Value" + "Data"."Yellow A_Value";
       "Data".TIme_LIGHT_A := "Data".Timer_Light_YellowA_Remain - "T1".ET;
   END_IF;
END_REGION

REGION Network 13
   RUNG wire#powerrail
      P_Contact(operand := "System Data"."Green A", bit := "Pulse3")
      Move(in := "Data"."Green A _Value", out1 => "Data".TIme_LIGHT_A)
   END_RUNG
   // the same network as SCL:
   #_w1 := "System Data"."Green A" AND NOT "Pulse3";   // rising edge of "System Data"."Green A"
   "Pulse3" := "System Data"."Green A";
   IF #_w1 THEN "Data".TIme_LIGHT_A := "Data"."Green A _Value"; END_IF;
END_REGION

REGION Network 14: GreenA
   RUNG wire#powerrail
      Contact( "System Data"."Green A" )
      { S7_Templates := "SrcType := DInt" } Sub(in1 := "Data"."Green A _Value", in2 := "T1".ET, out => "Data".TIme_LIGHT_A)
   END_RUNG
   // the same network as SCL:
   IF "System Data"."Green A" THEN "Data".TIme_LIGHT_A := "Data"."Green A _Value" - "T1".ET; END_IF;
END_REGION

REGION Network 15: Calculate Remain Time(In second) Light A
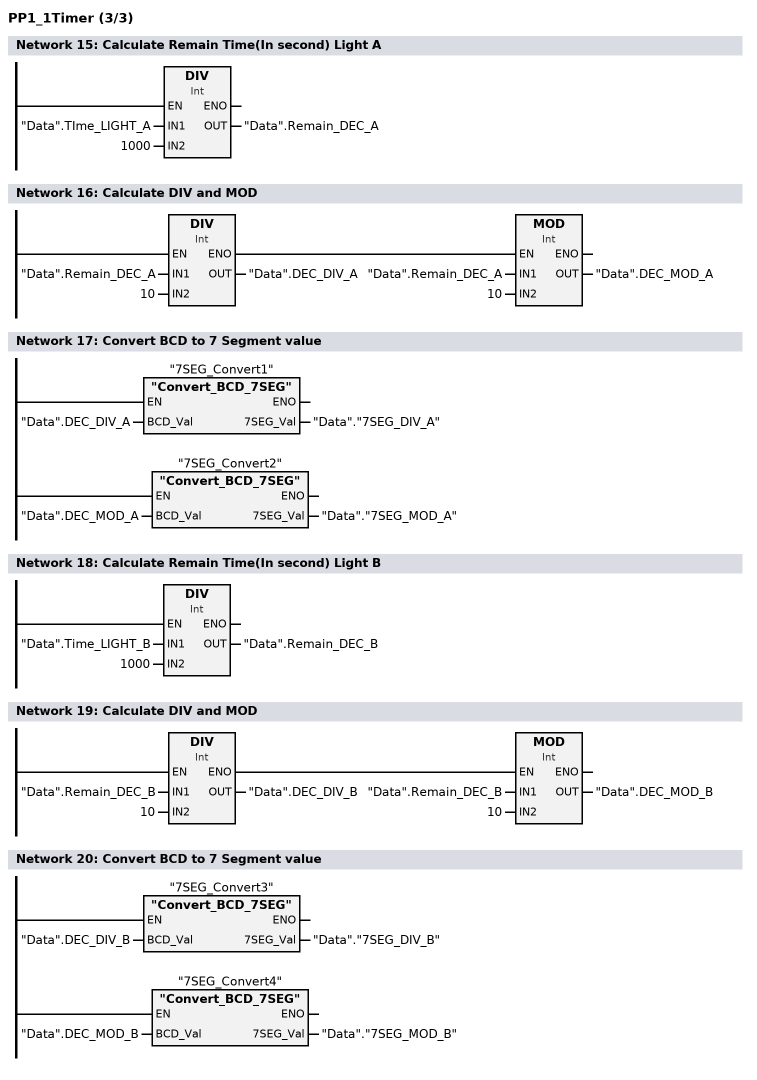
   RUNG wire#powerrail
      { S7_Templates := "SrcType := Int" } Div(in1 := "Data".TIme_LIGHT_A, in2 := 1000, out => "Data".Remain_DEC_A)
   END_RUNG
   // the same network as SCL:
   "Data".Remain_DEC_A := "Data".TIme_LIGHT_A / 1000;
END_REGION

REGION Network 16: Calculate DIV and MOD
   RUNG wire#powerrail
      { S7_Templates := "SrcType := Int" } Div(in1 := "Data".Remain_DEC_A, in2 := 10, out => "Data".DEC_DIV_A)
      { S7_Templates := "SrcType := Int" } Mod(in1 := "Data".Remain_DEC_A, in2 := 10, out => "Data".DEC_MOD_A)
   END_RUNG
   // the same network as SCL:
   "Data".DEC_DIV_A := "Data".Remain_DEC_A / 10;
   "Data".DEC_MOD_A := "Data".Remain_DEC_A MOD 10;
END_REGION

REGION Network 17: Convert BCD to 7 Segment value
   RUNG wire#powerrail
      "7SEG_Convert1"(BCD_Val := "Data".DEC_DIV_A, "7SEG_Val" => "Data"."7SEG_DIV_A")
   END_RUNG
   RUNG wire#powerrail
      "7SEG_Convert2"(BCD_Val := "Data".DEC_MOD_A, "7SEG_Val" => "Data"."7SEG_MOD_A")
   END_RUNG
   // the same network as SCL:
   "7SEG_Convert1"(BCD_Val := "Data".DEC_DIV_A, "7SEG_Val" => "Data"."7SEG_DIV_A");   // "Convert_BCD_7SEG"
   "7SEG_Convert2"(BCD_Val := "Data".DEC_MOD_A, "7SEG_Val" => "Data"."7SEG_MOD_A");   // "Convert_BCD_7SEG"
END_REGION

REGION Network 18: Calculate Remain Time(In second) Light B
   RUNG wire#powerrail
      { S7_Templates := "SrcType := Int" } Div(in1 := "Data".Time_LIGHT_B, in2 := 1000, out => "Data".Remain_DEC_B)
   END_RUNG
   // the same network as SCL:
   "Data".Remain_DEC_B := "Data".Time_LIGHT_B / 1000;
END_REGION

REGION Network 19: Calculate DIV and MOD
   RUNG wire#powerrail
      { S7_Templates := "SrcType := Int" } Div(in1 := "Data".Remain_DEC_B, in2 := 10, out => "Data".DEC_DIV_B)
      { S7_Templates := "SrcType := Int" } Mod(in1 := "Data".Remain_DEC_B, in2 := 10, out => "Data".DEC_MOD_B)
   END_RUNG
   // the same network as SCL:
   "Data".DEC_DIV_B := "Data".Remain_DEC_B / 10;
   "Data".DEC_MOD_B := "Data".Remain_DEC_B MOD 10;
END_REGION

REGION Network 20: Convert BCD to 7 Segment value
   RUNG wire#powerrail
      "7SEG_Convert3"(BCD_Val := "Data".DEC_DIV_B, "7SEG_Val" => "Data"."7SEG_DIV_B")
   END_RUNG
   RUNG wire#powerrail
      "7SEG_Convert4"(BCD_Val := "Data".DEC_MOD_B, "7SEG_Val" => "Data"."7SEG_MOD_B")
   END_RUNG
   // the same network as SCL:
   "7SEG_Convert3"(BCD_Val := "Data".DEC_DIV_B, "7SEG_Val" => "Data"."7SEG_DIV_B");   // "Convert_BCD_7SEG"
   "7SEG_Convert4"(BCD_Val := "Data".DEC_MOD_B, "7SEG_Val" => "Data"."7SEG_MOD_B");   // "Convert_BCD_7SEG"
END_REGION
END_FUNCTION

FUNCTION "PP3_Counter" : Void   // FC3, LAD
{ S7_Optimized_Access := 'TRUE' }
VERSION : 0.1
   VAR_TEMP   // added for the SCL form of the ladder/FBD networks
      _w1 : Bool;
   END_VAR
BEGIN

REGION Network 1: System
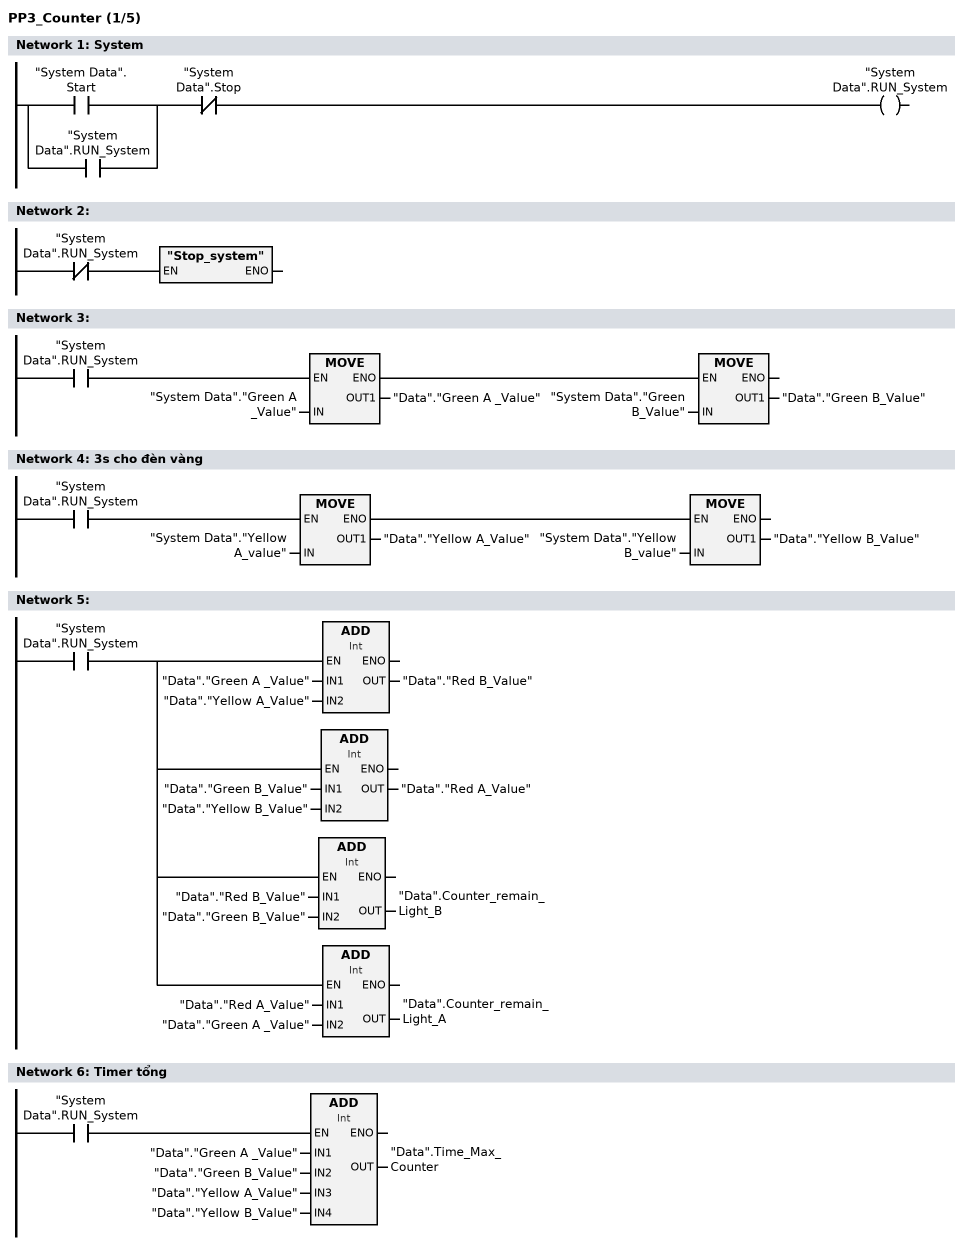
   RUNG wire#powerrail
      Contact( "System Data".Start )
      wire#w1
      I_Contact( "System Data".Stop )
      Coil( "System Data".RUN_System )
   END_RUNG
   RUNG wire#powerrail
      Contact( "System Data".RUN_System )
   END_RUNG wire#w1
   // the same network as SCL:
   "System Data".RUN_System := ("System Data".Start OR "System Data".RUN_System) AND NOT "System Data".Stop;
END_REGION

REGION Network 2
   RUNG wire#powerrail
      I_Contact( "System Data".RUN_System )
      "Stop_system"()
   END_RUNG
   // the same network as SCL:
   IF NOT "System Data".RUN_System THEN "Stop_system"(); END_IF;
END_REGION

REGION Network 3
   RUNG wire#powerrail
      Contact( "System Data".RUN_System )
      Move(in := "System Data"."Green A _Value", out1 => "Data"."Green A _Value")
      Move(in := "System Data"."Green B_Value", out1 => "Data"."Green B_Value")
   END_RUNG
   // the same network as SCL:
   IF "System Data".RUN_System THEN
       "Data"."Green A _Value" := "System Data"."Green A _Value";
       "Data"."Green B_Value" := "System Data"."Green B_Value";
   END_IF;
END_REGION

REGION Network 4: 3s cho đèn vàng
   RUNG wire#powerrail
      Contact( "System Data".RUN_System )
      Move(in := "System Data"."Yellow A_value", out1 => "Data"."Yellow A_Value")
      Move(in := "System Data"."Yellow B_value", out1 => "Data"."Yellow B_Value")
   END_RUNG
   // the same network as SCL:
   IF "System Data".RUN_System THEN
       "Data"."Yellow A_Value" := "System Data"."Yellow A_value";
       "Data"."Yellow B_Value" := "System Data"."Yellow B_value";
   END_IF;
END_REGION

REGION Network 5
   RUNG wire#powerrail
      Contact( "System Data".RUN_System )
      wire#w1
      { S7_Templates := "SrcType := Int" } Add(in1 := "Data"."Green A _Value", in2 := "Data"."Yellow A_Value", out => "Data"."Red B_Value")
   END_RUNG
   RUNG wire#w1
      { S7_Templates := "SrcType := Int" } Add(in1 := "Data"."Green B_Value", in2 := "Data"."Yellow B_Value", out => "Data"."Red A_Value")
   END_RUNG
   RUNG wire#w1
      { S7_Templates := "SrcType := Int" } Add(in1 := "Data"."Red B_Value", in2 := "Data"."Green B_Value", out => "Data".Counter_remain_Light_B)
   END_RUNG
   RUNG wire#w1
      { S7_Templates := "SrcType := Int" } Add(in1 := "Data"."Red A_Value", in2 := "Data"."Green A _Value", out => "Data".Counter_remain_Light_A)
   END_RUNG
   // the same network as SCL:
   IF "System Data".RUN_System THEN
       "Data"."Red B_Value" := "Data"."Green A _Value" + "Data"."Yellow A_Value";
       "Data"."Red A_Value" := "Data"."Green B_Value" + "Data"."Yellow B_Value";
       "Data".Counter_remain_Light_B := "Data"."Red B_Value" + "Data"."Green B_Value";
       "Data".Counter_remain_Light_A := "Data"."Red A_Value" + "Data"."Green A _Value";
   END_IF;
END_REGION

REGION Network 6: Timer tổng
   RUNG wire#powerrail
      Contact( "System Data".RUN_System )
      { S7_Templates := "SrcType := Int" } Add(in1 := "Data"."Green A _Value", in2 := "Data"."Green B_Value", in3 := "Data"."Yellow A_Value", in4 := "Data"."Yellow B_Value", out => "Data".Time_Max_Counter)
   END_RUNG
   // the same network as SCL:
   IF "System Data".RUN_System THEN
       "Data".Time_Max_Counter := "Data"."Green A _Value" + "Data"."Green B_Value" + "Data"."Yellow A_Value" + "Data"."Yellow B_Value";
   END_IF;
END_REGION

REGION Network 7: Tạo xung 1s
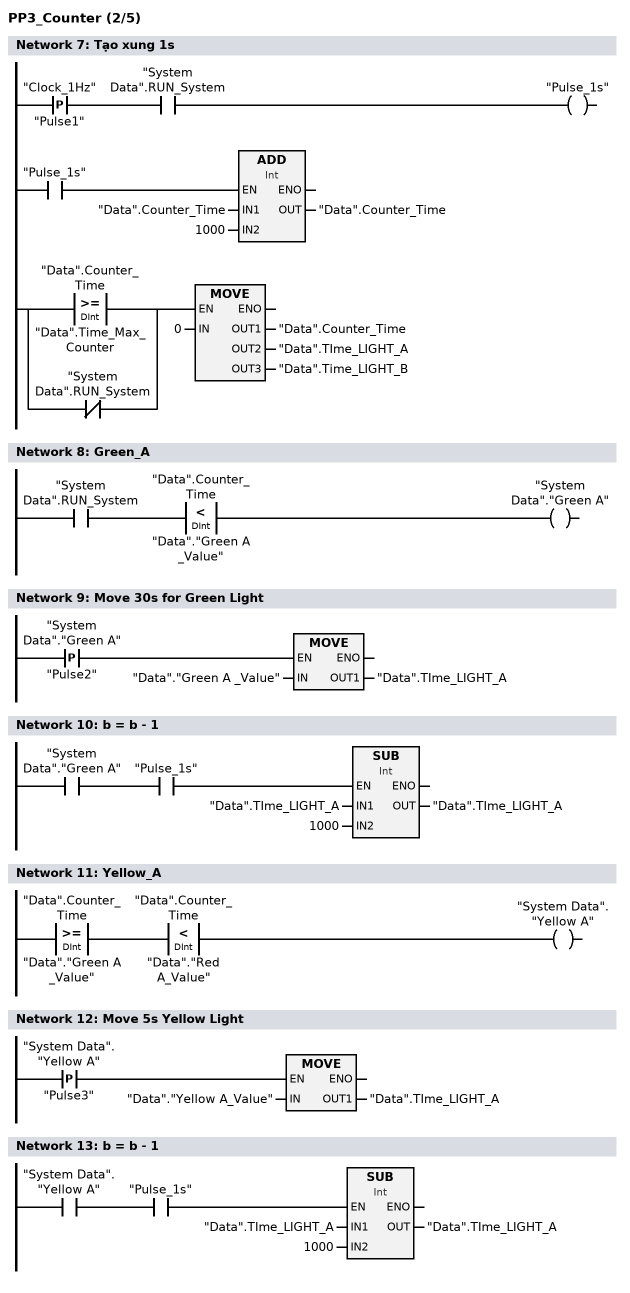
   RUNG wire#powerrail
      P_Contact(operand := "Clock_1Hz", bit := "Pulse1")
      Contact( "System Data".RUN_System )
      Coil( "Pulse_1s" )
   END_RUNG
   RUNG wire#powerrail
      Contact( "Pulse_1s" )
      { S7_Templates := "SrcType := Int" } Add(in1 := "Data".Counter_Time, in2 := 1000, out => "Data".Counter_Time)
   END_RUNG
   RUNG wire#powerrail
      { S7_Templates := "SrcType := DInt" } GE_Contact(in1 := "Data".Counter_Time, in2 := "Data".Time_Max_Counter)
      wire#w1
      Move(in := 0, out1 => "Data".Counter_Time, out2 => "Data".TIme_LIGHT_A, out3 => "Data".Time_LIGHT_B)
   END_RUNG
   RUNG wire#powerrail
      I_Contact( "System Data".RUN_System )
   END_RUNG wire#w1
   // the same network as SCL:
   #_w1 := "Clock_1Hz" AND NOT "Pulse1";   // rising edge of "Clock_1Hz"
   "Pulse1" := "Clock_1Hz";
   "Pulse_1s" := #_w1 AND "System Data".RUN_System;
   IF "Pulse_1s" THEN "Data".Counter_Time := "Data".Counter_Time + 1000; END_IF;
   IF ("Data".Counter_Time >= "Data".Time_Max_Counter) OR NOT "System Data".RUN_System THEN
       "Data".Counter_Time := 0;
       "Data".TIme_LIGHT_A := 0;
       "Data".Time_LIGHT_B := 0;
   END_IF;
END_REGION

REGION Network 8: Green_A
   RUNG wire#powerrail
      Contact( "System Data".RUN_System )
      { S7_Templates := "SrcType := DInt" } LT_Contact(in1 := "Data".Counter_Time, in2 := "Data"."Green A _Value")
      Coil( "System Data"."Green A" )
   END_RUNG
   // the same network as SCL:
   "System Data"."Green A" := "System Data".RUN_System AND ("Data".Counter_Time < "Data"."Green A _Value");
END_REGION

REGION Network 9: Move 30s for Green Light
   RUNG wire#powerrail
      P_Contact(operand := "System Data"."Green A", bit := "Pulse2")
      Move(in := "Data"."Green A _Value", out1 => "Data".TIme_LIGHT_A)
   END_RUNG
   // the same network as SCL:
   #_w1 := "System Data"."Green A" AND NOT "Pulse2";   // rising edge of "System Data"."Green A"
   "Pulse2" := "System Data"."Green A";
   IF #_w1 THEN "Data".TIme_LIGHT_A := "Data"."Green A _Value"; END_IF;
END_REGION

REGION Network 10: b = b - 1
   RUNG wire#powerrail
      Contact( "System Data"."Green A" )
      Contact( "Pulse_1s" )
      { S7_Templates := "SrcType := Int" } Sub(in1 := "Data".TIme_LIGHT_A, in2 := 1000, out => "Data".TIme_LIGHT_A)
   END_RUNG
   // the same network as SCL:
   IF "System Data"."Green A" AND "Pulse_1s" THEN "Data".TIme_LIGHT_A := "Data".TIme_LIGHT_A - 1000; END_IF;
END_REGION

REGION Network 11: Yellow_A
   RUNG wire#powerrail
      { S7_Templates := "SrcType := DInt" } GE_Contact(in1 := "Data".Counter_Time, in2 := "Data"."Green A _Value")
      { S7_Templates := "SrcType := DInt" } LT_Contact(in1 := "Data".Counter_Time, in2 := "Data"."Red A_Value")
      Coil( "System Data"."Yellow A" )
   END_RUNG
   // the same network as SCL:
   "System Data"."Yellow A" := ("Data".Counter_Time >= "Data"."Green A _Value") AND ("Data".Counter_Time < "Data"."Red A_Value");
END_REGION

REGION Network 12: Move 5s Yellow Light
   RUNG wire#powerrail
      P_Contact(operand := "System Data"."Yellow A", bit := "Pulse3")
      Move(in := "Data"."Yellow A_Value", out1 => "Data".TIme_LIGHT_A)
   END_RUNG
   // the same network as SCL:
   #_w1 := "System Data"."Yellow A" AND NOT "Pulse3";   // rising edge of "System Data"."Yellow A"
   "Pulse3" := "System Data"."Yellow A";
   IF #_w1 THEN "Data".TIme_LIGHT_A := "Data"."Yellow A_Value"; END_IF;
END_REGION

REGION Network 13: b = b - 1
   RUNG wire#powerrail
      Contact( "System Data"."Yellow A" )
      Contact( "Pulse_1s" )
      { S7_Templates := "SrcType := Int" } Sub(in1 := "Data".TIme_LIGHT_A, in2 := 1000, out => "Data".TIme_LIGHT_A)
   END_RUNG
   // the same network as SCL:
   IF "System Data"."Yellow A" AND "Pulse_1s" THEN "Data".TIme_LIGHT_A := "Data".TIme_LIGHT_A - 1000; END_IF;
END_REGION

REGION Network 14: Red_A
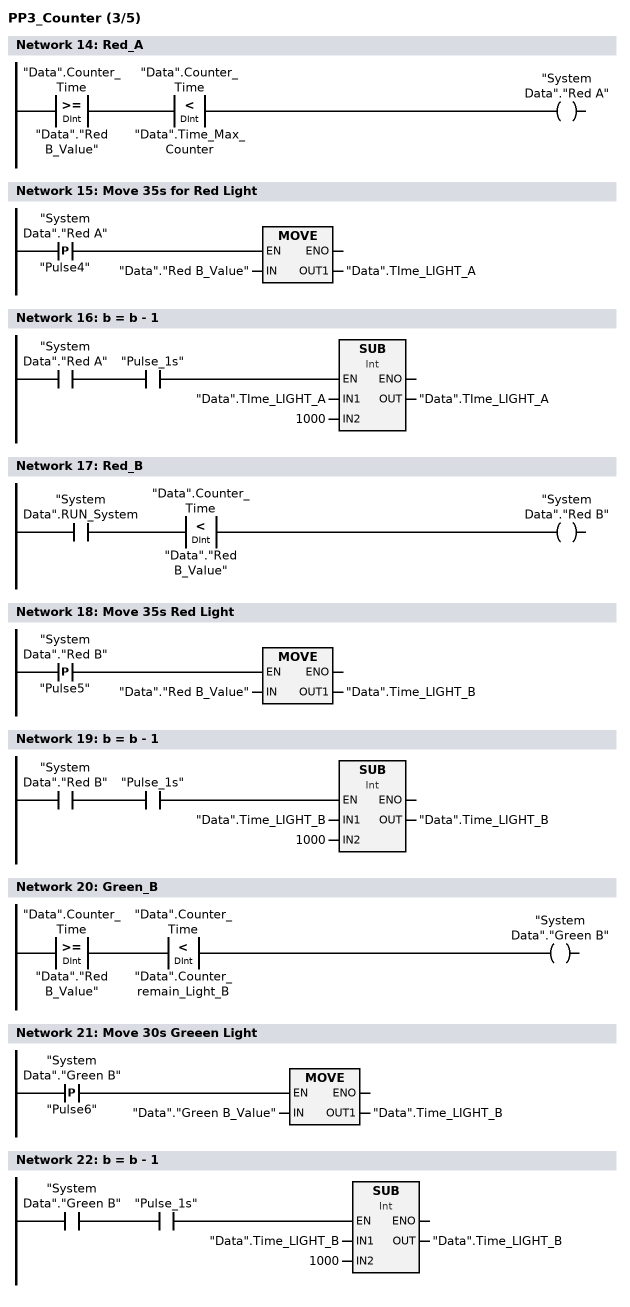
   RUNG wire#powerrail
      { S7_Templates := "SrcType := DInt" } GE_Contact(in1 := "Data".Counter_Time, in2 := "Data"."Red B_Value")
      { S7_Templates := "SrcType := DInt" } LT_Contact(in1 := "Data".Counter_Time, in2 := "Data".Time_Max_Counter)
      Coil( "System Data"."Red A" )
   END_RUNG
   // the same network as SCL:
   "System Data"."Red A" := ("Data".Counter_Time >= "Data"."Red B_Value") AND ("Data".Counter_Time < "Data".Time_Max_Counter);
END_REGION

REGION Network 15: Move 35s for Red Light
   RUNG wire#powerrail
      P_Contact(operand := "System Data"."Red A", bit := "Pulse4")
      Move(in := "Data"."Red B_Value", out1 => "Data".TIme_LIGHT_A)
   END_RUNG
   // the same network as SCL:
   #_w1 := "System Data"."Red A" AND NOT "Pulse4";   // rising edge of "System Data"."Red A"
   "Pulse4" := "System Data"."Red A";
   IF #_w1 THEN "Data".TIme_LIGHT_A := "Data"."Red B_Value"; END_IF;
END_REGION

REGION Network 16: b = b - 1
   RUNG wire#powerrail
      Contact( "System Data"."Red A" )
      Contact( "Pulse_1s" )
      { S7_Templates := "SrcType := Int" } Sub(in1 := "Data".TIme_LIGHT_A, in2 := 1000, out => "Data".TIme_LIGHT_A)
   END_RUNG
   // the same network as SCL:
   IF "System Data"."Red A" AND "Pulse_1s" THEN "Data".TIme_LIGHT_A := "Data".TIme_LIGHT_A - 1000; END_IF;
END_REGION

REGION Network 17: Red_B
   RUNG wire#powerrail
      Contact( "System Data".RUN_System )
      { S7_Templates := "SrcType := DInt" } LT_Contact(in1 := "Data".Counter_Time, in2 := "Data"."Red B_Value")
      Coil( "System Data"."Red B" )
   END_RUNG
   // the same network as SCL:
   "System Data"."Red B" := "System Data".RUN_System AND ("Data".Counter_Time < "Data"."Red B_Value");
END_REGION

REGION Network 18: Move 35s Red Light
   RUNG wire#powerrail
      P_Contact(operand := "System Data"."Red B", bit := "Pulse5")
      Move(in := "Data"."Red B_Value", out1 => "Data".Time_LIGHT_B)
   END_RUNG
   // the same network as SCL:
   #_w1 := "System Data"."Red B" AND NOT "Pulse5";   // rising edge of "System Data"."Red B"
   "Pulse5" := "System Data"."Red B";
   IF #_w1 THEN "Data".Time_LIGHT_B := "Data"."Red B_Value"; END_IF;
END_REGION

REGION Network 19: b = b - 1
   RUNG wire#powerrail
      Contact( "System Data"."Red B" )
      Contact( "Pulse_1s" )
      { S7_Templates := "SrcType := Int" } Sub(in1 := "Data".Time_LIGHT_B, in2 := 1000, out => "Data".Time_LIGHT_B)
   END_RUNG
   // the same network as SCL:
   IF "System Data"."Red B" AND "Pulse_1s" THEN "Data".Time_LIGHT_B := "Data".Time_LIGHT_B - 1000; END_IF;
END_REGION

REGION Network 20: Green_B
   RUNG wire#powerrail
      { S7_Templates := "SrcType := DInt" } GE_Contact(in1 := "Data".Counter_Time, in2 := "Data"."Red B_Value")
      { S7_Templates := "SrcType := DInt" } LT_Contact(in1 := "Data".Counter_Time, in2 := "Data".Counter_remain_Light_B)
      Coil( "System Data"."Green B" )
   END_RUNG
   // the same network as SCL:
   "System Data"."Green B" := ("Data".Counter_Time >= "Data"."Red B_Value") AND ("Data".Counter_Time < "Data".Counter_remain_Light_B);
END_REGION

REGION Network 21: Move 30s Greeen Light
   RUNG wire#powerrail
      P_Contact(operand := "System Data"."Green B", bit := "Pulse6")
      Move(in := "Data"."Green B_Value", out1 => "Data".Time_LIGHT_B)
   END_RUNG
   // the same network as SCL:
   #_w1 := "System Data"."Green B" AND NOT "Pulse6";   // rising edge of "System Data"."Green B"
   "Pulse6" := "System Data"."Green B";
   IF #_w1 THEN "Data".Time_LIGHT_B := "Data"."Green B_Value"; END_IF;
END_REGION

REGION Network 22: b = b - 1
   RUNG wire#powerrail
      Contact( "System Data"."Green B" )
      Contact( "Pulse_1s" )
      { S7_Templates := "SrcType := Int" } Sub(in1 := "Data".Time_LIGHT_B, in2 := 1000, out => "Data".Time_LIGHT_B)
   END_RUNG
   // the same network as SCL:
   IF "System Data"."Green B" AND "Pulse_1s" THEN "Data".Time_LIGHT_B := "Data".Time_LIGHT_B - 1000; END_IF;
END_REGION

REGION Network 23: Yellow_B
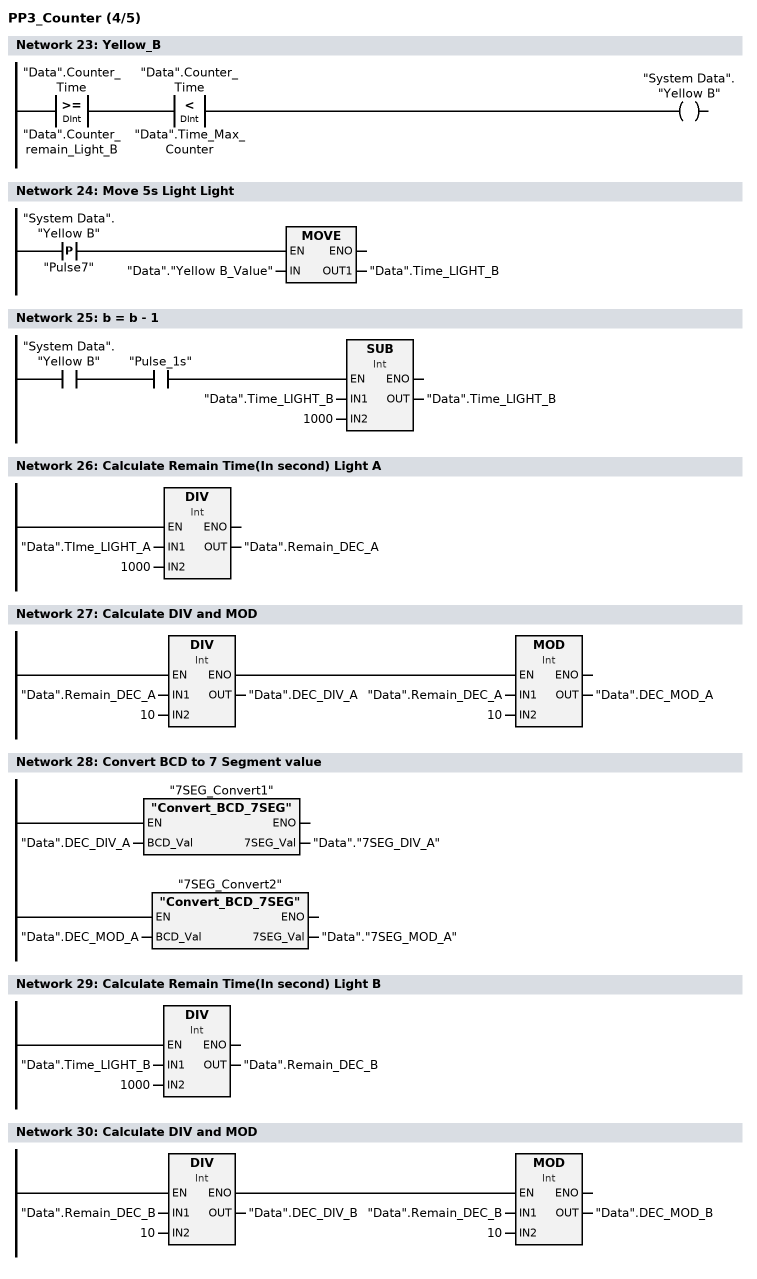
   RUNG wire#powerrail
      { S7_Templates := "SrcType := DInt" } GE_Contact(in1 := "Data".Counter_Time, in2 := "Data".Counter_remain_Light_B)
      { S7_Templates := "SrcType := DInt" } LT_Contact(in1 := "Data".Counter_Time, in2 := "Data".Time_Max_Counter)
      Coil( "System Data"."Yellow B" )
   END_RUNG
   // the same network as SCL:
   "System Data"."Yellow B" := ("Data".Counter_Time >= "Data".Counter_remain_Light_B) AND ("Data".Counter_Time < "Data".Time_Max_Counter);
END_REGION

REGION Network 24: Move 5s Light Light
   RUNG wire#powerrail
      P_Contact(operand := "System Data"."Yellow B", bit := "Pulse7")
      Move(in := "Data"."Yellow B_Value", out1 => "Data".Time_LIGHT_B)
   END_RUNG
   // the same network as SCL:
   #_w1 := "System Data"."Yellow B" AND NOT "Pulse7";   // rising edge of "System Data"."Yellow B"
   "Pulse7" := "System Data"."Yellow B";
   IF #_w1 THEN "Data".Time_LIGHT_B := "Data"."Yellow B_Value"; END_IF;
END_REGION

REGION Network 25: b = b - 1
   RUNG wire#powerrail
      Contact( "System Data"."Yellow B" )
      Contact( "Pulse_1s" )
      { S7_Templates := "SrcType := Int" } Sub(in1 := "Data".Time_LIGHT_B, in2 := 1000, out => "Data".Time_LIGHT_B)
   END_RUNG
   // the same network as SCL:
   IF "System Data"."Yellow B" AND "Pulse_1s" THEN "Data".Time_LIGHT_B := "Data".Time_LIGHT_B - 1000; END_IF;
END_REGION

REGION Network 26: Calculate Remain Time(In second) Light A
   RUNG wire#powerrail
      { S7_Templates := "SrcType := Int" } Div(in1 := "Data".TIme_LIGHT_A, in2 := 1000, out => "Data".Remain_DEC_A)
   END_RUNG
   // the same network as SCL:
   "Data".Remain_DEC_A := "Data".TIme_LIGHT_A / 1000;
END_REGION

REGION Network 27: Calculate DIV and MOD
   RUNG wire#powerrail
      { S7_Templates := "SrcType := Int" } Div(in1 := "Data".Remain_DEC_A, in2 := 10, out => "Data".DEC_DIV_A)
      { S7_Templates := "SrcType := Int" } Mod(in1 := "Data".Remain_DEC_A, in2 := 10, out => "Data".DEC_MOD_A)
   END_RUNG
   // the same network as SCL:
   "Data".DEC_DIV_A := "Data".Remain_DEC_A / 10;
   "Data".DEC_MOD_A := "Data".Remain_DEC_A MOD 10;
END_REGION

REGION Network 28: Convert BCD to 7 Segment value
   RUNG wire#powerrail
      "7SEG_Convert1"(BCD_Val := "Data".DEC_DIV_A, "7SEG_Val" => "Data"."7SEG_DIV_A")
   END_RUNG
   RUNG wire#powerrail
      "7SEG_Convert2"(BCD_Val := "Data".DEC_MOD_A, "7SEG_Val" => "Data"."7SEG_MOD_A")
   END_RUNG
   // the same network as SCL:
   "7SEG_Convert1"(BCD_Val := "Data".DEC_DIV_A, "7SEG_Val" => "Data"."7SEG_DIV_A");   // "Convert_BCD_7SEG"
   "7SEG_Convert2"(BCD_Val := "Data".DEC_MOD_A, "7SEG_Val" => "Data"."7SEG_MOD_A");   // "Convert_BCD_7SEG"
END_REGION

REGION Network 29: Calculate Remain Time(In second) Light B
   RUNG wire#powerrail
      { S7_Templates := "SrcType := Int" } Div(in1 := "Data".Time_LIGHT_B, in2 := 1000, out => "Data".Remain_DEC_B)
   END_RUNG
   // the same network as SCL:
   "Data".Remain_DEC_B := "Data".Time_LIGHT_B / 1000;
END_REGION

REGION Network 30: Calculate DIV and MOD
   RUNG wire#powerrail
      { S7_Templates := "SrcType := Int" } Div(in1 := "Data".Remain_DEC_B, in2 := 10, out => "Data".DEC_DIV_B)
      { S7_Templates := "SrcType := Int" } Mod(in1 := "Data".Remain_DEC_B, in2 := 10, out => "Data".DEC_MOD_B)
   END_RUNG
   // the same network as SCL:
   "Data".DEC_DIV_B := "Data".Remain_DEC_B / 10;
   "Data".DEC_MOD_B := "Data".Remain_DEC_B MOD 10;
END_REGION

REGION Network 31: Convert BCD to 7 Segment value
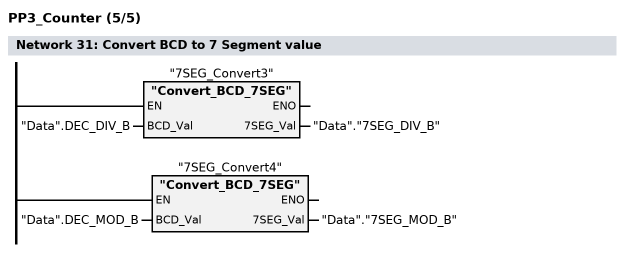
   RUNG wire#powerrail
      "7SEG_Convert3"(BCD_Val := "Data".DEC_DIV_B, "7SEG_Val" => "Data"."7SEG_DIV_B")
   END_RUNG
   RUNG wire#powerrail
      "7SEG_Convert4"(BCD_Val := "Data".DEC_MOD_B, "7SEG_Val" => "Data"."7SEG_MOD_B")
   END_RUNG
   // the same network as SCL:
   "7SEG_Convert3"(BCD_Val := "Data".DEC_DIV_B, "7SEG_Val" => "Data"."7SEG_DIV_B");   // "Convert_BCD_7SEG"
   "7SEG_Convert4"(BCD_Val := "Data".DEC_MOD_B, "7SEG_Val" => "Data"."7SEG_MOD_B");   // "Convert_BCD_7SEG"
END_REGION
END_FUNCTION

FUNCTION "Light_night" : Void   // FC4, LAD
{ S7_Optimized_Access := 'TRUE' }
VERSION : 0.1
BEGIN

REGION Network 1
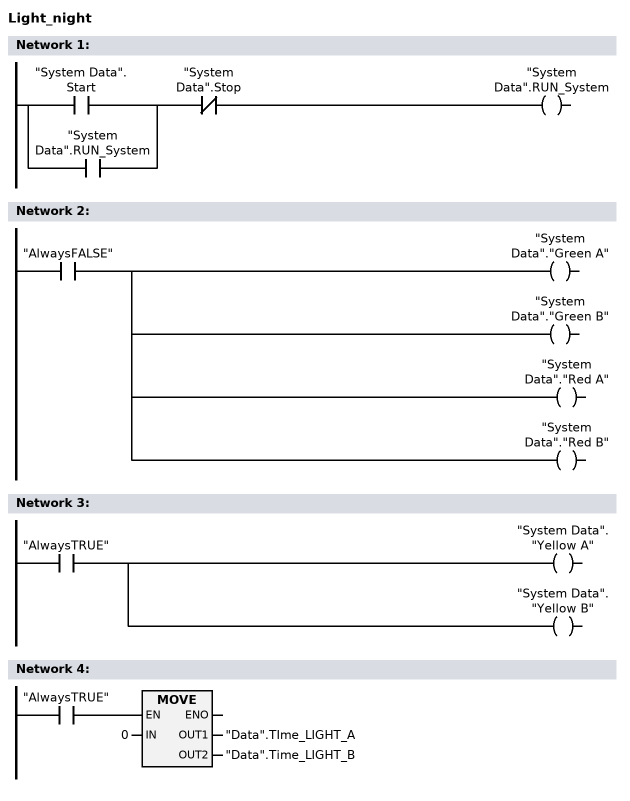
   RUNG wire#powerrail
      Contact( "System Data".Start )
      wire#w1
      I_Contact( "System Data".Stop )
      Coil( "System Data".RUN_System )
   END_RUNG
   RUNG wire#powerrail
      Contact( "System Data".RUN_System )
   END_RUNG wire#w1
   // the same network as SCL:
   "System Data".RUN_System := ("System Data".Start OR "System Data".RUN_System) AND NOT "System Data".Stop;
END_REGION

REGION Network 2
   RUNG wire#powerrail
      Contact( "AlwaysFALSE" )
      wire#w1
      Coil( "System Data"."Green A" )
   END_RUNG
   RUNG wire#w1
      Coil( "System Data"."Green B" )
   END_RUNG
   RUNG wire#w1
      Coil( "System Data"."Red A" )
   END_RUNG
   RUNG wire#w1
      Coil( "System Data"."Red B" )
   END_RUNG
   // the same network as SCL:
   "System Data"."Green A" := "AlwaysFALSE";
   "System Data"."Green B" := "AlwaysFALSE";
   "System Data"."Red A" := "AlwaysFALSE";
   "System Data"."Red B" := "AlwaysFALSE";
END_REGION

REGION Network 3
   RUNG wire#powerrail
      Contact( "AlwaysTRUE" )
      wire#w1
      Coil( "System Data"."Yellow A" )
   END_RUNG
   RUNG wire#w1
      Coil( "System Data"."Yellow B" )
   END_RUNG
   // the same network as SCL:
   "System Data"."Yellow A" := "AlwaysTRUE";
   "System Data"."Yellow B" := "AlwaysTRUE";
END_REGION

REGION Network 4
   RUNG wire#powerrail
      Contact( "AlwaysTRUE" )
      Move(in := 0, out1 => "Data".TIme_LIGHT_A, out2 => "Data".Time_LIGHT_B)
   END_RUNG
   // the same network as SCL:
   IF "AlwaysTRUE" THEN
       "Data".TIme_LIGHT_A := 0;
       "Data".Time_LIGHT_B := 0;
   END_IF;
END_REGION
END_FUNCTION

FUNCTION "Function Local time" : Void   // FC5, LAD
{ S7_Optimized_Access := 'TRUE' }
VERSION : 0.1
BEGIN

REGION Network 1: Function read local time
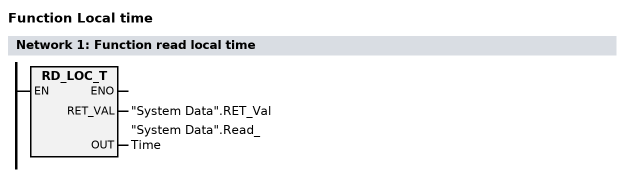
   "System Data".RET_Val := RD_LOC_T(OUT => "System Data".Read_Time);
END_REGION
END_FUNCTION

FUNCTION "Stop_system" : Void   // FC6, LAD
{ S7_Optimized_Access := 'TRUE' }
VERSION : 0.1
BEGIN

REGION Network 1
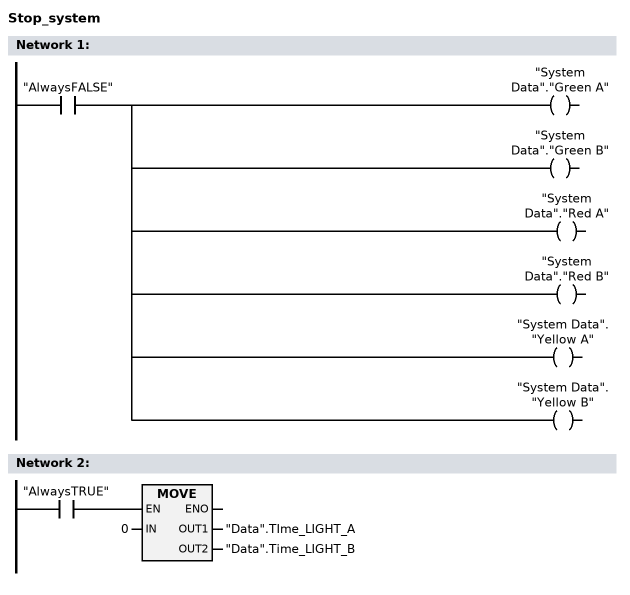
   RUNG wire#powerrail
      Contact( "AlwaysFALSE" )
      wire#w1
      Coil( "System Data"."Green A" )
   END_RUNG
   RUNG wire#w1
      Coil( "System Data"."Green B" )
   END_RUNG
   RUNG wire#w1
      Coil( "System Data"."Red A" )
   END_RUNG
   RUNG wire#w1
      Coil( "System Data"."Red B" )
   END_RUNG
   RUNG wire#w1
      Coil( "System Data"."Yellow A" )
   END_RUNG
   RUNG wire#w1
      Coil( "System Data"."Yellow B" )
   END_RUNG
   // the same network as SCL:
   "System Data"."Green A" := "AlwaysFALSE";
   "System Data"."Green B" := "AlwaysFALSE";
   "System Data"."Red A" := "AlwaysFALSE";
   "System Data"."Red B" := "AlwaysFALSE";
   "System Data"."Yellow A" := "AlwaysFALSE";
   "System Data"."Yellow B" := "AlwaysFALSE";
END_REGION

REGION Network 2
   RUNG wire#powerrail
      Contact( "AlwaysTRUE" )
      Move(in := 0, out1 => "Data".TIme_LIGHT_A, out2 => "Data".Time_LIGHT_B)
   END_RUNG
   // the same network as SCL:
   IF "AlwaysTRUE" THEN
       "Data".TIme_LIGHT_A := 0;
       "Data".Time_LIGHT_B := 0;
   END_IF;
END_REGION
END_FUNCTION

FUNCTION "Output_mapping" : Void   // FC7, LAD
{ S7_Optimized_Access := 'TRUE' }
VERSION : 0.1
BEGIN

REGION Network 1: LightA
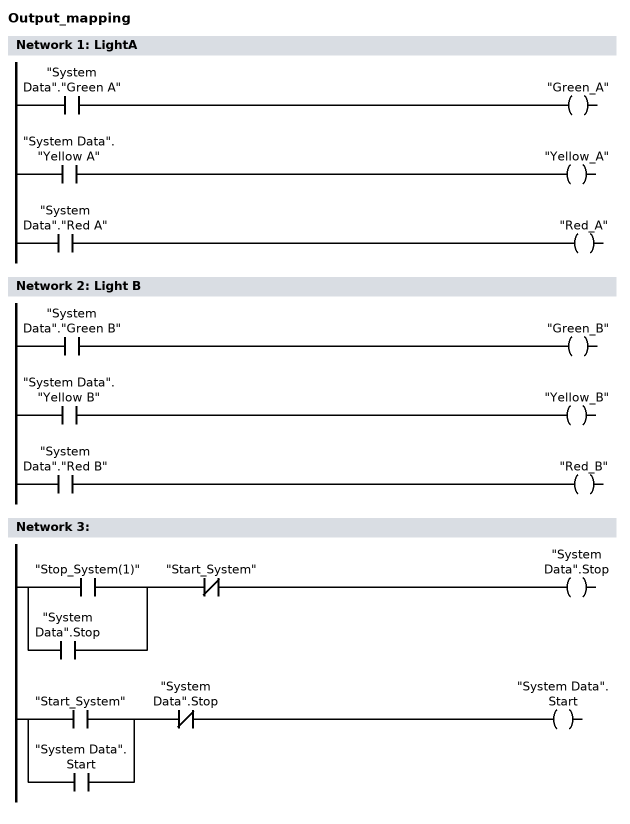
   RUNG wire#powerrail
      Contact( "System Data"."Green A" )
      Coil( "Green_A" )
   END_RUNG
   RUNG wire#powerrail
      Contact( "System Data"."Yellow A" )
      Coil( "Yellow_A" )
   END_RUNG
   RUNG wire#powerrail
      Contact( "System Data"."Red A" )
      Coil( "Red_A" )
   END_RUNG
   // the same network as SCL:
   "Green_A" := "System Data"."Green A";
   "Yellow_A" := "System Data"."Yellow A";
   "Red_A" := "System Data"."Red A";
END_REGION

REGION Network 2: Light B
   RUNG wire#powerrail
      Contact( "System Data"."Green B" )
      Coil( "Green_B" )
   END_RUNG
   RUNG wire#powerrail
      Contact( "System Data"."Yellow B" )
      Coil( "Yellow_B" )
   END_RUNG
   RUNG wire#powerrail
      Contact( "System Data"."Red B" )
      Coil( "Red_B" )
   END_RUNG
   // the same network as SCL:
   "Green_B" := "System Data"."Green B";
   "Yellow_B" := "System Data"."Yellow B";
   "Red_B" := "System Data"."Red B";
END_REGION

REGION Network 3
   RUNG wire#powerrail
      Contact( "Stop_System(1)" )
      wire#w1
      I_Contact( "Start_System" )
      Coil( "System Data".Stop )
   END_RUNG
   RUNG wire#powerrail
      Contact( "System Data".Stop )
   END_RUNG wire#w1
   RUNG wire#powerrail
      Contact( "Start_System" )
      wire#w2
      I_Contact( "System Data".Stop )
      Coil( "System Data".Start )
   END_RUNG
   RUNG wire#powerrail
      Contact( "System Data".Start )
   END_RUNG wire#w2
   // the same network as SCL:
   "System Data".Stop := ("Stop_System(1)" OR "System Data".Stop) AND NOT "Start_System";
   "System Data".Start := ("Start_System" OR "System Data".Start) AND NOT "System Data".Stop;
END_REGION
END_FUNCTION

FUNCTION "Emergency" : Void   // FC8, LAD
{ S7_Optimized_Access := 'TRUE' }
VERSION : 0.1
BEGIN

REGION Network 1
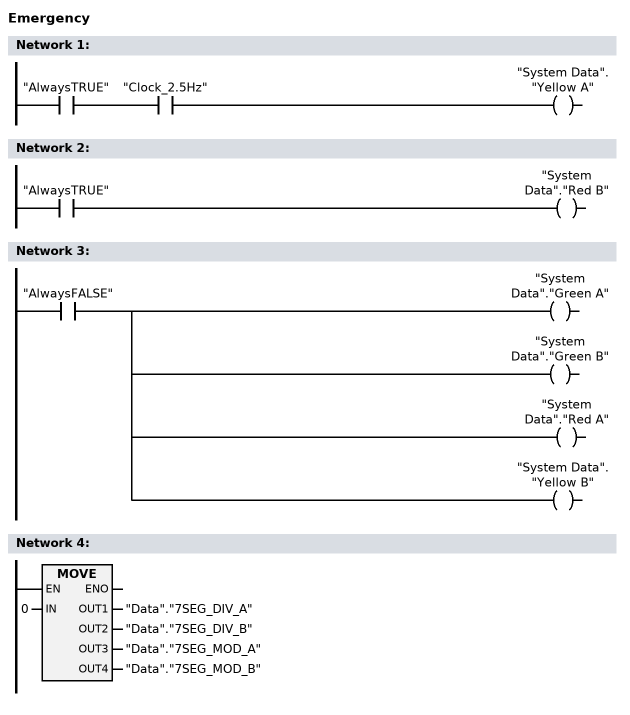
   RUNG wire#powerrail
      Contact( "AlwaysTRUE" )
      Contact( "Clock_2.5Hz" )
      Coil( "System Data"."Yellow A" )
   END_RUNG
   // the same network as SCL:
   "System Data"."Yellow A" := "AlwaysTRUE" AND "Clock_2.5Hz";
END_REGION

REGION Network 2
   RUNG wire#powerrail
      Contact( "AlwaysTRUE" )
      Coil( "System Data"."Red B" )
   END_RUNG
   // the same network as SCL:
   "System Data"."Red B" := "AlwaysTRUE";
END_REGION

REGION Network 3
   RUNG wire#powerrail
      Contact( "AlwaysFALSE" )
      wire#w1
      Coil( "System Data"."Green A" )
   END_RUNG
   RUNG wire#w1
      Coil( "System Data"."Green B" )
   END_RUNG
   RUNG wire#w1
      Coil( "System Data"."Red A" )
   END_RUNG
   RUNG wire#w1
      Coil( "System Data"."Yellow B" )
   END_RUNG
   // the same network as SCL:
   "System Data"."Green A" := "AlwaysFALSE";
   "System Data"."Green B" := "AlwaysFALSE";
   "System Data"."Red A" := "AlwaysFALSE";
   "System Data"."Yellow B" := "AlwaysFALSE";
END_REGION

REGION Network 4
   RUNG wire#powerrail
      Move(in := 0, out1 => "Data"."7SEG_DIV_A", out2 => "Data"."7SEG_DIV_B", out3 => "Data"."7SEG_MOD_A", out4 => "Data"."7SEG_MOD_B")
   END_RUNG
   // the same network as SCL:
   "Data"."7SEG_DIV_A" := 0;
   "Data"."7SEG_DIV_B" := 0;
   "Data"."7SEG_MOD_A" := 0;
   "Data"."7SEG_MOD_B" := 0;
END_REGION
END_FUNCTION

ORGANIZATION_BLOCK "Main"   // OB1, LAD, ProgramCycle
TITLE = "Main Program Sweep (Cycle)"
{ S7_Optimized_Access := 'TRUE' }
VERSION : 0.1
   VAR_INPUT
      Initial_Call : Bool;   // Initial call of this OB
      Remanence : Bool;   // =True, if remanent data are available
   END_VAR
   VAR_TEMP   // added for the SCL form of the ladder/FBD networks
      _w1 : Bool;
      _w2 : Bool;
      _w3 : Bool;
   END_VAR
BEGIN

REGION Network 1: Read local time
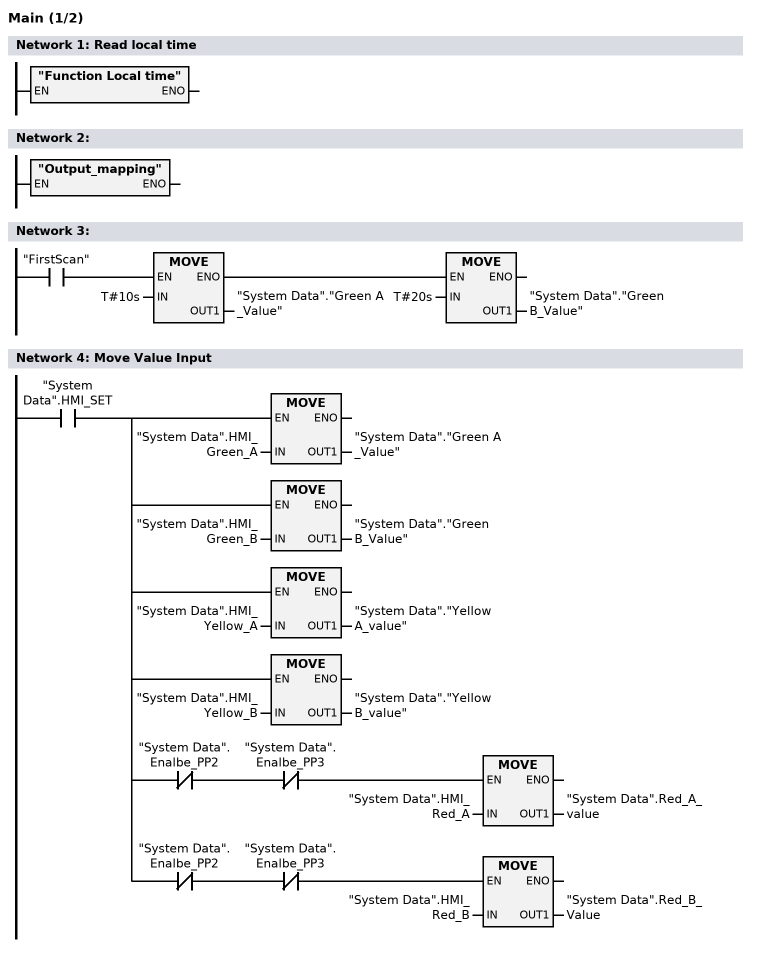
   RUNG wire#powerrail
      "Function Local time"()
   END_RUNG
   // the same network as SCL:
   "Function Local time"();
END_REGION

REGION Network 2
   RUNG wire#powerrail
      "Output_mapping"()
   END_RUNG
   // the same network as SCL:
   "Output_mapping"();
END_REGION

REGION Network 3
   RUNG wire#powerrail
      Contact( "FirstScan" )
      Move(in := T#10s, out1 => "System Data"."Green A _Value")
      Move(in := T#20s, out1 => "System Data"."Green B_Value")
   END_RUNG
   // the same network as SCL:
   IF "FirstScan" THEN
       "System Data"."Green A _Value" := T#10s;
       "System Data"."Green B_Value" := T#20s;
   END_IF;
END_REGION

REGION Network 4: Move Value Input
   RUNG wire#powerrail
      Contact( "System Data".HMI_SET )
      wire#w1
      Move(in := "System Data".HMI_Green_A, out1 => "System Data"."Green A _Value")
   END_RUNG
   RUNG wire#w1
      Move(in := "System Data".HMI_Green_B, out1 => "System Data"."Green B_Value")
   END_RUNG
   RUNG wire#w1
      Move(in := "System Data".HMI_Yellow_A, out1 => "System Data"."Yellow A_value")
   END_RUNG
   RUNG wire#w1
      Move(in := "System Data".HMI_Yellow_B, out1 => "System Data"."Yellow B_value")
   END_RUNG
   RUNG wire#w1
      I_Contact( "System Data".Enalbe_PP2 )
      I_Contact( "System Data".Enalbe_PP3 )
      Move(in := "System Data".HMI_Red_A, out1 => "System Data".Red_A_value)
   END_RUNG
   RUNG wire#w1
      I_Contact( "System Data".Enalbe_PP2 )
      I_Contact( "System Data".Enalbe_PP3 )
      Move(in := "System Data".HMI_Red_B, out1 => "System Data".Red_B_Value)
   END_RUNG
   // the same network as SCL:
   IF "System Data".HMI_SET THEN
       "System Data"."Green A _Value" := "System Data".HMI_Green_A;
       "System Data"."Green B_Value" := "System Data".HMI_Green_B;
       "System Data"."Yellow A_value" := "System Data".HMI_Yellow_A;
       "System Data"."Yellow B_value" := "System Data".HMI_Yellow_B;
   END_IF;
   IF "System Data".HMI_SET AND NOT "System Data".Enalbe_PP2 AND NOT "System Data".Enalbe_PP3 THEN
       "System Data".Red_A_value := "System Data".HMI_Red_A;
       "System Data".Red_B_Value := "System Data".HMI_Red_B;
   END_IF;
END_REGION

REGION Network 5
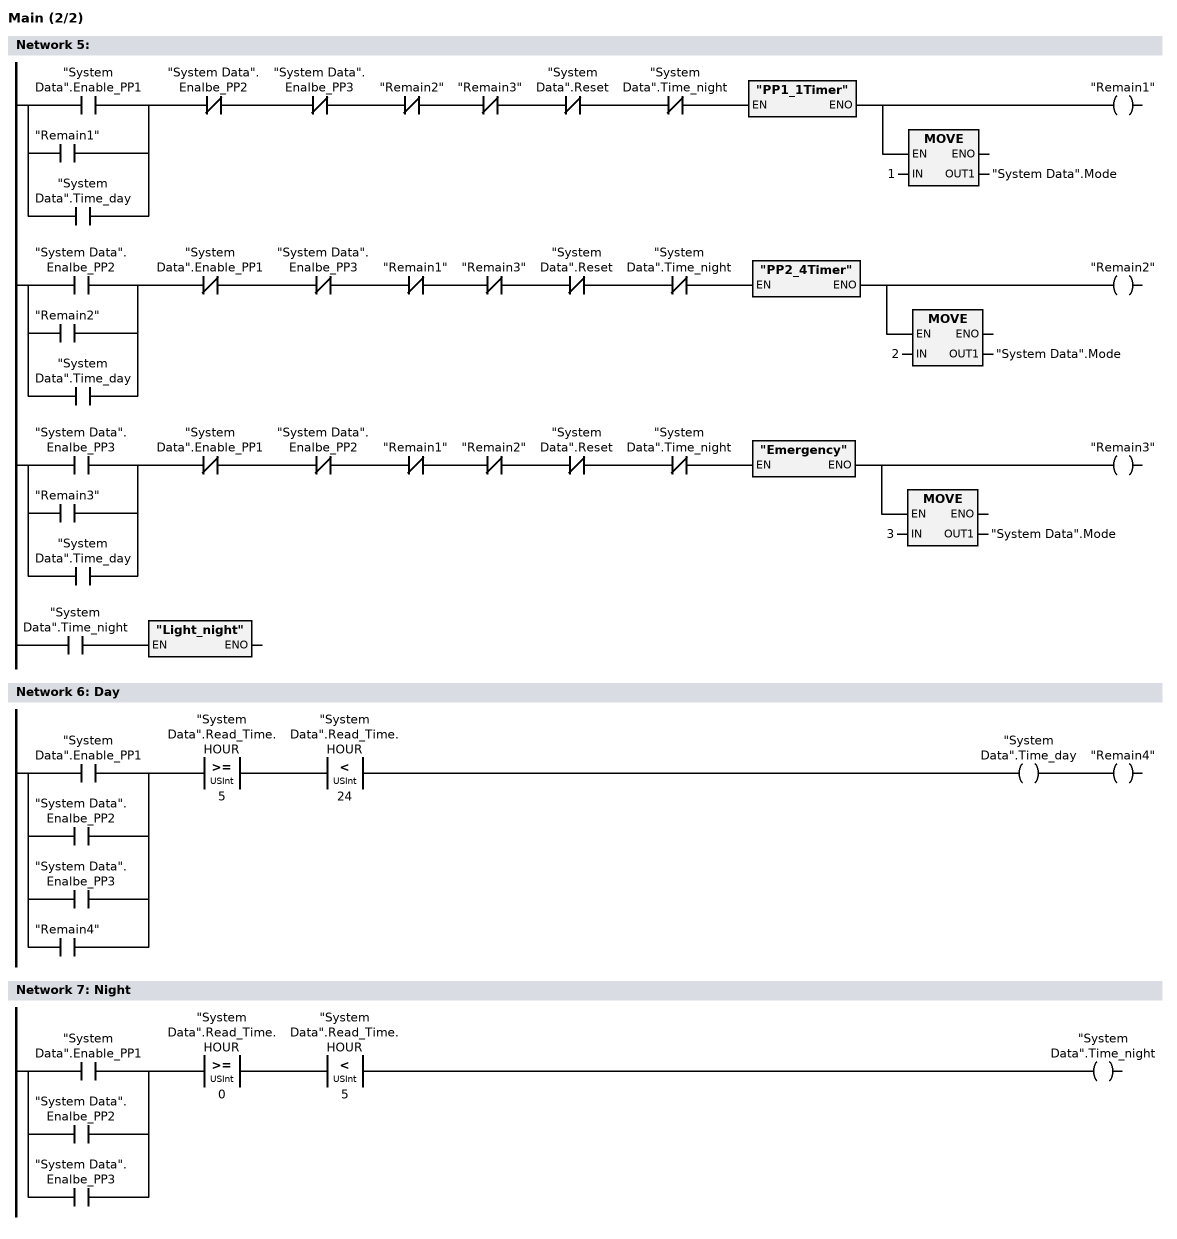
   RUNG wire#powerrail
      Contact( "System Data".Enable_PP1 )
      wire#w1
      I_Contact( "System Data".Enalbe_PP2 )
      I_Contact( "System Data".Enalbe_PP3 )
      I_Contact( "Remain2" )
      I_Contact( "Remain3" )
      I_Contact( "System Data".Reset )
      I_Contact( "System Data".Time_night )
      "PP1_1Timer"()
      wire#w2
      Coil( "Remain1" )
   END_RUNG
   RUNG wire#powerrail
      Contact( "Remain1" )
   END_RUNG wire#w1
   RUNG wire#powerrail
      Contact( "System Data".Time_day )
   END_RUNG wire#w1
   RUNG wire#w2
      Move(in := 1, out1 => "System Data".Mode)
   END_RUNG
   RUNG wire#powerrail
      Contact( "System Data".Enalbe_PP2 )
      wire#w3
      I_Contact( "System Data".Enable_PP1 )
      I_Contact( "System Data".Enalbe_PP3 )
      I_Contact( "Remain1" )
      I_Contact( "Remain3" )
      I_Contact( "System Data".Reset )
      I_Contact( "System Data".Time_night )
      "PP2_4Timer"()
      wire#w4
      Coil( "Remain2" )
   END_RUNG
   RUNG wire#powerrail
      Contact( "Remain2" )
   END_RUNG wire#w3
   RUNG wire#powerrail
      Contact( "System Data".Time_day )
   END_RUNG wire#w3
   RUNG wire#w4
      Move(in := 2, out1 => "System Data".Mode)
   END_RUNG
   RUNG wire#powerrail
      Contact( "System Data".Enalbe_PP3 )
      wire#w5
      I_Contact( "System Data".Enable_PP1 )
      I_Contact( "System Data".Enalbe_PP2 )
      I_Contact( "Remain1" )
      I_Contact( "Remain2" )
      I_Contact( "System Data".Reset )
      I_Contact( "System Data".Time_night )
      "Emergency"()
      wire#w6
      Coil( "Remain3" )
   END_RUNG
   RUNG wire#powerrail
      Contact( "Remain3" )
   END_RUNG wire#w5
   RUNG wire#powerrail
      Contact( "System Data".Time_day )
   END_RUNG wire#w5
   RUNG wire#w6
      Move(in := 3, out1 => "System Data".Mode)
   END_RUNG
   RUNG wire#powerrail
      Contact( "System Data".Time_night )
      "Light_night"()
   END_RUNG
   // the same network as SCL:
   "PP1_1Timer"(EN := ("System Data".Enable_PP1 OR "Remain1" OR "System Data".Time_day) AND NOT "System Data".Enalbe_PP2 AND NOT "System Data".Enalbe_PP3 AND NOT "Remain2" AND NOT "Remain3" AND NOT "System Data".Reset AND NOT "System Data".Time_night,
                ENO => #_w1);
   "Remain1" := #_w1;
   IF #_w1 THEN "System Data".Mode := 1; END_IF;
   "PP2_4Timer"(EN := ("System Data".Enalbe_PP2 OR "Remain2" OR "System Data".Time_day) AND NOT "System Data".Enable_PP1 AND NOT "System Data".Enalbe_PP3 AND NOT "Remain1" AND NOT "Remain3" AND NOT "System Data".Reset AND NOT "System Data".Time_night,
                ENO => #_w2);
   "Remain2" := #_w2;
   IF #_w2 THEN "System Data".Mode := 2; END_IF;
   "Emergency"(EN := ("System Data".Enalbe_PP3 OR "Remain3" OR "System Data".Time_day) AND NOT "System Data".Enable_PP1 AND NOT "System Data".Enalbe_PP2 AND NOT "Remain1" AND NOT "Remain2" AND NOT "System Data".Reset AND NOT "System Data".Time_night,
               ENO => #_w3);
   "Remain3" := #_w3;
   IF #_w3 THEN "System Data".Mode := 3; END_IF;
   IF "System Data".Time_night THEN "Light_night"(); END_IF;
END_REGION

REGION Network 6: Day
   RUNG wire#powerrail
      Contact( "System Data".Enable_PP1 )
      wire#w1
      { S7_Templates := "SrcType := USInt" } GE_Contact(in1 := "System Data".Read_Time.HOUR, in2 := 5)
      { S7_Templates := "SrcType := USInt" } LT_Contact(in1 := "System Data".Read_Time.HOUR, in2 := 24)
      Coil( "System Data".Time_day )
      Coil( "Remain4" )
   END_RUNG
   RUNG wire#powerrail
      Contact( "System Data".Enalbe_PP2 )
   END_RUNG wire#w1
   RUNG wire#powerrail
      Contact( "System Data".Enalbe_PP3 )
   END_RUNG wire#w1
   RUNG wire#powerrail
      Contact( "Remain4" )
   END_RUNG wire#w1
   // the same network as SCL:
   "System Data".Time_day := ("System Data".Enable_PP1 OR "System Data".Enalbe_PP2 OR "System Data".Enalbe_PP3 OR "Remain4") AND ("System Data".Read_Time.HOUR >= 5) AND ("System Data".Read_Time.HOUR < 24);
   "Remain4" := "System Data".Time_day;
END_REGION

REGION Network 7: Night
   RUNG wire#powerrail
      Contact( "System Data".Enable_PP1 )
      wire#w1
      { S7_Templates := "SrcType := USInt" } GE_Contact(in1 := "System Data".Read_Time.HOUR, in2 := 0)
      { S7_Templates := "SrcType := USInt" } LT_Contact(in1 := "System Data".Read_Time.HOUR, in2 := 5)
      Coil( "System Data".Time_night )
   END_RUNG
   RUNG wire#powerrail
      Contact( "System Data".Enalbe_PP2 )
   END_RUNG wire#w1
   RUNG wire#powerrail
      Contact( "System Data".Enalbe_PP3 )
   END_RUNG wire#w1
   // the same network as SCL:
   "System Data".Time_night := ("System Data".Enable_PP1 OR "System Data".Enalbe_PP2 OR "System Data".Enalbe_PP3) AND ("System Data".Read_Time.HOUR >= 0) AND ("System Data".Read_Time.HOUR < 5);
END_REGION
END_ORGANIZATION_BLOCK

(* ===== HMI "HMI_RT_1" =====
system functions are stored by id; their names below are inferred from use
connection "HMI_Connection_6": ETHERNET, SMART_S7_1500_OMS

HMI tags "Default tag table"
   "Data_TIme_LIGHT_A" : DInt = PLC Data.TIme_LIGHT_A AT %DB1.DBD0, 1 s
   "Data_Time_LIGHT_B" : DInt = PLC Data.Time_LIGHT_B AT %DB1.DBD0, 1 s
   "Data_7SEG_DIV" : Byte = PLC Data.7SEG_DIV_A AT %DB1.DBB0, 1 s
   "Data_7SEG_DIV_B" : Byte = PLC Data.7SEG_DIV_B AT %DB1.DBB0, 1 s
   "Data_7SEG_MOD" : Byte = PLC Data.7SEG_MOD_A AT %DB1.DBB0, 1 s
   "Data_7SEG_MOD_B" : Byte = PLC Data.7SEG_MOD_B AT %DB1.DBB0, 1 s
   "Data_Timer_Red A_Value" : DInt = PLC Data."Red A_Value" AT %DB1.DBD0, 1 s
   "Data_Timer_Red B_Value" : DInt = PLC Data."Red B_Value" AT %DB1.DBD0, 1 s
   "System Data_Cancel" : Bool = PLC "System Data".Reset AT %DB1.DBX0.0, 1 s
   "System Data_Enable_PP1" : Bool = PLC "System Data".Enable_PP1 AT %DB1.DBX0.0, 1 s
   "System Data_Enalbe_PP2" : Bool = PLC "System Data".Enalbe_PP2 AT %DB1.DBX0.0, 1 s
   "System Data_Enalbe_PP3" : Bool = PLC "System Data".Enalbe_PP3 AT %DB1.DBX0.0, 1 s
   "System Data_Red A" : Bool = PLC "System Data"."Red A" AT %DB1.DBX0.0, 1 s
   "System Data_Yellow A" : Bool = PLC "System Data"."Yellow A" AT %DB1.DBX0.0, 1 s
   "System Data_Green A" : Bool = PLC "System Data"."Green A" AT %DB1.DBX0.0, 1 s
   "System Data_Green B" : Bool = PLC "System Data"."Green B" AT %DB1.DBX0.0, 1 s
   "System Data_Yellow B" : Bool = PLC "System Data"."Yellow B" AT %DB1.DBX0.0, 1 s
   "System Data_Red B" : Bool = PLC "System Data"."Red B" AT %DB1.DBX0.0, 1 s
   "System Data_Stop" : Bool = PLC "System Data".Stop AT %DB1.DBX0.0, 1 s
   "System Data_Start" : Bool = PLC "System Data".Start AT %DB1.DBX0.0, 1 s
   "System Data_Visible" : Bool = PLC "System Data".Visible_1, 1 s
   "System Data_HMI_Red_A" : DInt = PLC "System Data".HMI_Red_A, 1 s
   "System Data_HMI_Green_A" : DInt = PLC "System Data".HMI_Green_A, 1 s
   "System Data_HMI_Yellow_A" : DInt = PLC "System Data".HMI_Yellow_A, 1 s
   "System Data_HMI_SET" : Bool = PLC "System Data".HMI_SET, 1 s
   "Data_DEC_DIV_A" : Int = PLC Data.Remain_DEC_A, 1 s
   "Data_DEC_DIV_B" : Int = PLC Data.Remain_DEC_B, 1 s
   "System Data_HMI_Green_B" : DInt = PLC "System Data".HMI_Green_B, 1 s
   "System Data_HMI_Yellow_B" : DInt = PLC "System Data".HMI_Yellow_B, 1 s
   "System Data_Visible_2" : Bool = PLC "System Data".Visible_2, 1 s
   "System Data_Mode" : DInt = PLC "System Data".Mode, 1 s

text list "Light_mode": 1 '1 Light'; 2 '2 Light'; 3 'Emergency'; 0 'Stop'

Template "Template_1" 800x480
   Button "Exit" at 714,429 size 71x50; TextOff 'Exit'; PictureOff "ExitRuntime_KTP700_Basic_PN_TR"; PictureOn "ExitRuntime_KTP700_Basic_PN_TR"
      on Release: StopRuntime(0)
   Button "Template_Button" at 614,429 size 71x50; TextOff 'Text'
   Button "Template_Button_1" at 514,429 size 71x50; TextOff 'Text'
   Button "Template_Button_2" at 414,429 size 71x50; TextOff 'Text'
   Button "Template_Button_3" at 314,429 size 71x50; TextOff 'Text'
   Button "Template_Button_4" at 214,429 size 71x50; TextOff 'Text'
   Button "Alarms" at 114,429 size 71x50; TextOff 'Alarms'; PictureOff "AlarmDisplay_KTP700_Basic_PN_TR"; PictureOn "AlarmDisplay_KTP700_Basic_PN_TR"
      on Release: function_ef3f5d25("Alarm window_Unacknowledged", -1)
   Button "Start screen" at 14,429 size 71x50; TextOff 'Start screen'; PictureOff "NavigateHome_KTP700_Basic_PN_TR"; PictureOn "NavigateHome_KTP700_Basic_PN_TR"
      on Release: ActivateScreen("Root screen", 0)
   DateTimeField "HmiScreenItemData" at 695,25 size 105x25
   DateTimeField "HmiScreenItemData_1" at 695,0 size 105x25
   GraphicView "Logo" at 0,0 size 91x51; Picture "Logo of HMI_1"

screen "Root screen" 800x480, template "Template_1"
   GraphicView "Graphic view_5" at 91,0 size 72x111; Picture "Graphic_9"
   GraphicView "Graphic view_7" at 167,424 size 64x43; Picture "Graphic_10"
   GraphicView "Graphic view_8" at 18,331 size 75x125; Picture "Graphic_11"
   GraphicView "Graphic view_3" at 38,387 size 142x90; Picture "Graphic_3"
   GraphicView "Graphic view_4" at 56,63 size 176x95; Picture "Graphic_6"
   GraphicView "Graphic view_12" at 573,48 size 227x62; Picture "Graphic_14"
   GraphicView "Graphic view_2" at 556,40 size 130x105; Picture "Graphic_2"
   GraphicView "Graphic view_11" at 680,36 size 120x105; Picture "Graphic_2"
   GraphicView "Graphic view_13" at 0,0 size 70x95; Picture "Graphic_15"
   GraphicView "Graphic view_6" at 156,45 size 74x63; Picture "Graphic_1"
   GraphicView "Graphic view_16" at 2,430 size 54x47; Picture "Graphic_16"
   GraphicView "Graphic view_18" at 476,43 size 35x46; Picture "Graphic_17"
   GraphicView "Graphic view_19" at 496,3 size 35x46; Picture "Graphic_17"
   GraphicView "Graphic view_20" at 510,41 size 35x46; Picture "Graphic_17"
   GraphicView "Graphic view_21" at 713,127 size 35x46; Picture "Graphic_17"
   GraphicView "Graphic view_22" at 465,3 size 35x46; Picture "Graphic_17"
   GraphicView "Graphic view_23" at 753,128 size 35x46; Picture "Graphic_17"
   GraphicView "Graphic view_25" at 663,189 size 100x38; Picture "Graphic_19"
   GraphicView "Graphic view_26" at 333,4 size 42x49; Picture "Graphic_20"
   GraphicView "Graphic view_27" at 54,245 size 127x47; Picture "Graphic_22"
   Group "Group_3" at 466,147 size 94x32
   Group "Group_4" at 212,309 size 94x32
   GraphicView "Graphic view_1" at 85,338 size 86x64; Picture "Graphic_3"
   Group "Group_5" at 465,298 size 32x94
   Group "Group_2" at 274,69 size 32x94
   GraphicView "Graphic view_10" at 244,129 size 30x35; Picture "Graphic_12"
   GraphicView "Graphic view_9" at 10,100 size 49x61; Picture "Graphic_12"
   Group "Group_6" at 264,31 size 41x37
   Group "Group_7" at 468,109 size 43x37
   Group "Group_8" at 258,344 size 43x37
   Group "Group_9" at 498,299 size 41x37
   Group "Group_10" at 574,380 size 223x97
   Group "Group_1" at 515,273 size 285x205
   Group "Group" at 547,341 size 253x135
   GraphicView "Graphic view_14" at 545,189 size 100x38; Picture "Graphic_19"
   GraphicView "Graphic view_15" at 179,366 size 86x64; Picture "Graphic_3"
   GraphicView "Graphic view_17" at 678,128 size 35x46; Picture "Graphic_17"
   Circle "Circle_8" at 277,102 size 26x26
      Appearance <- "System Data_Yellow B"
   Circle "Circle_7" at 277,71 size 26x26
      Appearance <- "System Data_Green B"
   Circle "Circle_9" at 277,134 size 26x26
      Appearance <- "System Data_Red B"
   Circle "Circle_11" at 468,331 size 26x26
      Appearance <- "System Data_Yellow B"
   Circle "Circle_12" at 468,363 size 26x26
      Appearance <- "System Data_Red B"
   Circle "Circle_10" at 468,300 size 26x26
      Appearance <- "System Data_Green B"
   Circle "Circle_4" at 277,312 size 26x26
      Appearance <- "System Data_Green A"
   Circle "Circle_5" at 246,312 size 26x26
      Appearance <- "System Data_Yellow A"
   Circle "Circle_6" at 215,312 size 26x26
      Appearance <- "System Data_Red A"
   Circle "Circle_1" at 469,150 size 26x26
      Appearance <- "System Data_Green A"
   Circle "Circle_2" at 500,150 size 26x26
      Appearance <- "System Data_Yellow A"
   Circle "Circle_3" at 532,150 size 26x26
      Appearance <- "System Data_Red A"
   Rectangle "Rectangle_28" at 549,341 size 249x135
      Visibility <- "System Data_Visible"
   Button "Button_3" at 721,450 size 78x26; TextOff 'SET'
      on Release: ResetBit("System Data_HMI_SET")
      on Press: SetBit("System Data_HMI_SET")
      Visibility <- "System Data_Visible"
   Button "Button_4" at 721,397 size 79x26; TextOff 'Start'
      on Release: ResetBit("System Data_Start")
      on Press: SetBit("System Data_Start")
      Visibility <- "System Data_Visible"
   Button "Button_2" at 721,423 size 78x26; TextOff 'Stop'
      on Release: ResetBit("System Data_Stop")
      on Press: SetBit("System Data_Stop")
      Visibility <- "System Data_Visible"
   Button "Button_5" at 711,341 size 88x27; TextOff 'X'
      on Click: InvertBit("System Data_Visible")
      Visibility <- "System Data_Visible"
   TextField "Text field_5" at 555,345 size 66x17; Text 'LIGHT'
      Visibility <- "System Data_Visible"
   TextField "Text field_6" at 547,387 size 66x18; Text 'Green'
      Visibility <- "System Data_Visible"
   TextField "Text field_7" at 547,420 size 66x18; Text 'Yellow'
      Visibility <- "System Data_Visible"
   TextField "Text field_8" at 548,445 size 66x18; Text 'Red'
      Visibility <- "System Data_Visible"
   IOField "I/O field_4" at 614,417 size 83x24; FormatPattern 99
      ProcessValue <- "System Data_HMI_Yellow_A"
      Visibility <- "System Data_Visible"
   IOField "I/O field_3" at 614,386 size 83x24; FormatPattern 99
      ProcessValue <- "System Data_HMI_Green_A"
      Visibility <- "System Data_Visible"
   IOField "I/O field_5" at 614,444 size 83x24; FormatPattern 99
      ProcessValue <- "System Data_HMI_Red_A"
      Visibility <- "System Data_Visible"
   Rectangle "Rectangle_31" at 289,31 size 13x4
      Appearance <- "Data_7SEG_MOD_B"
   Rectangle "Rectangle_45" at 301,35 size 4x14
      Appearance <- "Data_7SEG_MOD_B"
   Rectangle "Rectangle_46" at 289,48 size 13x4
      Appearance <- "Data_7SEG_MOD_B"
   Rectangle "Rectangle_47" at 301,51 size 4x14
      Appearance <- "Data_7SEG_MOD_B"
   Rectangle "Rectangle_48" at 289,64 size 13x4
      Appearance <- "Data_7SEG_MOD_B"
   Rectangle "Rectangle_49" at 286,51 size 4x14
      Appearance <- "Data_7SEG_MOD_B"
   Rectangle "Rectangle_50" at 286,35 size 4x14
      Appearance <- "Data_7SEG_MOD_B"
   Rectangle "Rectangle_51" at 267,31 size 14x4
      Appearance <- "Data_7SEG_DIV_B"
   Rectangle "Rectangle_52" at 280,35 size 4x14
      Appearance <- "Data_7SEG_DIV_B"
   Rectangle "Rectangle_53" at 267,48 size 14x4
      Appearance <- "Data_7SEG_DIV_B"
   Rectangle "Rectangle_54" at 280,51 size 4x14
      Appearance <- "Data_7SEG_DIV_B"
   Rectangle "Rectangle_55" at 267,64 size 14x4
      Appearance <- "Data_7SEG_DIV_B"
   Rectangle "Rectangle_56" at 264,51 size 4x14
      Appearance <- "Data_7SEG_DIV_B"
   Rectangle "Rectangle_57" at 264,35 size 4x14
      Appearance <- "Data_7SEG_DIV_B"
   Rectangle "Rectangle_58" at 494,109 size 14x4
      Appearance <- "Data_7SEG_MOD"
   Rectangle "Rectangle_59" at 507,113 size 4x14
      Appearance <- "Data_7SEG_MOD"
   Rectangle "Rectangle_60" at 494,126 size 14x4
      Appearance <- "Data_7SEG_MOD"
   Rectangle "Rectangle_61" at 507,129 size 4x14
      Appearance <- "Data_7SEG_MOD"
   Rectangle "Rectangle_62" at 494,142 size 14x4
      Appearance <- "Data_7SEG_MOD"
   Rectangle "Rectangle_63" at 491,129 size 4x13
      Appearance <- "Data_7SEG_MOD"
   Rectangle "Rectangle_64" at 491,113 size 4x14
      Appearance <- "Data_7SEG_MOD"
   Rectangle "Rectangle_65" at 471,109 size 14x4
      Appearance <- "Data_7SEG_DIV"
   Rectangle "Rectangle_66" at 484,113 size 4x14
      Appearance <- "Data_7SEG_DIV"
   Rectangle "Rectangle_67" at 471,126 size 14x4
      Appearance <- "Data_7SEG_DIV"
   Rectangle "Rectangle_68" at 484,129 size 4x14
      Appearance <- "Data_7SEG_DIV"
   Rectangle "Rectangle_69" at 471,142 size 14x4
      Appearance <- "Data_7SEG_DIV"
   Rectangle "Rectangle_70" at 468,129 size 4x14
      Appearance <- "Data_7SEG_DIV"
   Rectangle "Rectangle_71" at 468,113 size 4x14
      Appearance <- "Data_7SEG_DIV"
   Rectangle "Rectangle_72" at 284,344 size 14x4
      Appearance <- "Data_7SEG_MOD"
   Rectangle "Rectangle_73" at 297,348 size 4x14
      Appearance <- "Data_7SEG_MOD"
   Rectangle "Rectangle_74" at 284,361 size 14x4
      Appearance <- "Data_7SEG_MOD"
   Rectangle "Rectangle_75" at 297,364 size 4x14
      Appearance <- "Data_7SEG_MOD"
   Rectangle "Rectangle_76" at 284,377 size 14x4
      Appearance <- "Data_7SEG_MOD"
   Rectangle "Rectangle_77" at 281,364 size 4x13
      Appearance <- "Data_7SEG_MOD"
   Rectangle "Rectangle_78" at 281,348 size 4x14
      Appearance <- "Data_7SEG_MOD"
   Rectangle "Rectangle_79" at 261,344 size 14x4
      Appearance <- "Data_7SEG_DIV"
   Rectangle "Rectangle_80" at 274,348 size 4x14
      Appearance <- "Data_7SEG_DIV"
   Rectangle "Rectangle_81" at 261,361 size 14x4
      Appearance <- "Data_7SEG_DIV"
   Rectangle "Rectangle_82" at 274,364 size 4x14
      Appearance <- "Data_7SEG_DIV"
   Rectangle "Rectangle_83" at 261,377 size 14x4
      Appearance <- "Data_7SEG_DIV"
   Rectangle "Rectangle_84" at 258,364 size 4x14
      Appearance <- "Data_7SEG_DIV"
   Rectangle "Rectangle_85" at 258,348 size 4x14
      Appearance <- "Data_7SEG_DIV"
   Rectangle "Rectangle_86" at 523,299 size 13x4
      Appearance <- "Data_7SEG_MOD_B"
   Rectangle "Rectangle_87" at 535,303 size 4x14
      Appearance <- "Data_7SEG_MOD_B"
   Rectangle "Rectangle_88" at 523,316 size 13x4
      Appearance <- "Data_7SEG_MOD_B"
   Rectangle "Rectangle_89" at 535,319 size 4x14
      Appearance <- "Data_7SEG_MOD_B"
   Rectangle "Rectangle_90" at 523,332 size 13x4
      Appearance <- "Data_7SEG_MOD_B"
   Rectangle "Rectangle_91" at 520,319 size 4x14
      Appearance <- "Data_7SEG_MOD_B"
   Rectangle "Rectangle_92" at 520,303 size 4x14
      Appearance <- "Data_7SEG_MOD_B"
   Rectangle "Rectangle_93" at 501,299 size 14x4
      Appearance <- "Data_7SEG_DIV_B"
   Rectangle "Rectangle_94" at 514,303 size 4x14
      Appearance <- "Data_7SEG_DIV_B"
   Rectangle "Rectangle_95" at 501,316 size 14x4
      Appearance <- "Data_7SEG_DIV_B"
   Rectangle "Rectangle_96" at 514,319 size 4x14
      Appearance <- "Data_7SEG_DIV_B"
   Rectangle "Rectangle_97" at 501,332 size 14x4
      Appearance <- "Data_7SEG_DIV_B"
   Rectangle "Rectangle_98" at 498,319 size 4x14
      Appearance <- "Data_7SEG_DIV_B"
   Rectangle "Rectangle_99" at 498,303 size 4x14
      Appearance <- "Data_7SEG_DIV_B"
   TextField "Text field_3" at 574,382 size 106x22; Text 'Control Panel'
   Button "Button_6" at 690,381 size 107x32; TextOff '1 Light'
      on Click: InvertBit("System Data_Visible")
      on Release: ResetBit("System Data_Enable_PP1")
      on Press: SetBit("System Data_Enable_PP1")
      Appearance <- "System Data_Enable_PP1"
   Button "Button_7" at 690,413 size 106x32; TextOff '2 Light'
      on Click: InvertBit("System Data_Visible_2")
      on Release: ResetBit("System Data_Enalbe_PP2")
      on Press: SetBit("System Data_Enalbe_PP2")
      Appearance <- "System Data_Enalbe_PP2"
   Button "Button_9" at 690,445 size 106x32; TextOff 'Emergency'
      on Release: ResetBit("System Data_Enalbe_PP3")
      on Press: SetBit("System Data_Enalbe_PP3")
      Appearance <- "System Data_Enalbe_PP3"
   SymbolicIOField "Symbolic I/O field_1" at 574,445 size 118x32; TextOn '1'; TextOff '0'; TextList "Light_mode"
      ProcessValue <- "System Data_Mode"
   Rectangle "Rectangle_38" at 517,273 size 282x205
      Visibility <- "System Data_Visible_2"
   Rectangle "Rectangle_39" at 517,302 size 134x142
      Visibility <- "System Data_Visible_2"
   IOField "I/O field_1" at 579,329 size 67x30; FormatPattern 99
      Visibility <- "System Data_Visible_2"
      ProcessValue <- "System Data_HMI_Green_A"
   IOField "I/O field_2" at 579,365 size 67x30; FormatPattern 99
      Visibility <- "System Data_Visible_2"
      ProcessValue <- "System Data_HMI_Yellow_A"
   IOField "I/O field_6" at 579,402 size 67x30; FormatPattern 99
      Visibility <- "System Data_Visible_2"
      ProcessValue <- "Data_Timer_Red A_Value"
   Button "Button_11" at 726,448 size 73x30; TextOff 'SET'
      on Release: ResetBit("System Data_HMI_SET")
      on Press: SetBit("System Data_HMI_SET")
      Visibility <- "System Data_Visible_2"
   Button "Button_12" at 517,449 size 79x29; TextOff 'Start'
      on Release: ResetBit("System Data_Start")
      on Press: SetBit("System Data_Start")
      Visibility <- "System Data_Visible_2"
   TextField "Text field_9" at 515,298 size 66x26; Text 'Light A'
      Visibility <- "System Data_Visible_2"
   Rectangle "Rectangle_40" at 664,301 size 134x142
      Visibility <- "System Data_Visible_2"
   IOField "I/O field_9" at 726,326 size 67x29; FormatPattern 99
      Visibility <- "System Data_Visible_2"
      ProcessValue <- "System Data_HMI_Green_B"
   IOField "I/O field_10" at 726,364 size 67x29; FormatPattern 99
      Visibility <- "System Data_Visible_2"
      ProcessValue <- "System Data_HMI_Yellow_B"
   IOField "I/O field_11" at 726,401 size 67x29; FormatPattern 99
      Visibility <- "System Data_Visible_2"
      ProcessValue <- "Data_Timer_Red B_Value"
   TextField "Text field_10" at 663,296 size 66x29; Text 'Light B'
      Visibility <- "System Data_Visible_2"
   TextField "Text field_1" at 520,334 size 56x27; Text 'Green'
      Visibility <- "System Data_Visible_2"
   TextField "Text field_2" at 522,365 size 56x27; Text 'Yellow'
      Visibility <- "System Data_Visible_2"
   TextField "Text field_13" at 519,401 size 56x27; Text 'Red'
      Visibility <- "System Data_Visible_2"
   TextField "Text field_14" at 667,328 size 56x26; Text 'Green'
      Visibility <- "System Data_Visible_2"
   TextField "Text field_15" at 670,364 size 56x26; Text 'Yellow'
      Visibility <- "System Data_Visible_2"
   TextField "Text field_16" at 664,400 size 56x26; Text 'Red'
      Visibility <- "System Data_Visible_2"
   Button "Button_14" at 722,274 size 78x27; TextOff 'X'
      on Click: InvertBit("System Data_Visible_2")
      Visibility <- "System Data_Visible_2"
   Button "Button_15" at 595,449 size 78x29; TextOff 'Stop'
      on Release: ResetBit("System Data_Stop")
      on Press: SetBit("System Data_Stop")
      Appearance <- "System Data_Stop"
      Visibility <- "System Data_Visible_2"

screen "Screen_1" 800x480
   Rectangle "Rectangle_53" at 577,275 size 221x135
      Visibility <- "System Data_Visible"
   Button "Button_2" at 730,384 size 69x26; TextOff 'SET'
      on Release: ResetBit("System Data_HMI_SET")
      on Press: SetBit("System Data_HMI_SET")
      Visibility <- "System Data_Visible"
   Button "Button_5" at 730,331 size 70x26; TextOff 'Start'
      on Release: ResetBit("System Data_Start")
      on Press: SetBit("System Data_Start")
      Visibility <- "System Data_Visible"
   Button "Button_6" at 730,357 size 69x26; TextOff 'Reset'
      on Release: ResetBit("System Data_Stop")
      on Press: SetBit("System Data_Stop")
      Visibility <- "System Data_Visible"
   Button "Button_7" at 721,275 size 78x27; TextOff 'X'
      on Click: InvertBit("System Data_Visible")
      Visibility <- "System Data_Visible"
   TextField "Text field_1" at 582,279 size 59x17; Text 'LIGHT'
      Visibility <- "System Data_Visible"
   TextField "Text field_2" at 575,321 size 59x18; Text 'Green'
      Visibility <- "System Data_Visible"
   TextField "Text field_11" at 575,354 size 59x18; Text 'Yellow'
      Visibility <- "System Data_Visible"
   TextField "Text field_12" at 576,379 size 59x18; Text 'Red'
      Visibility <- "System Data_Visible"
   IOField "I/O field_1" at 635,348 size 74x24; FormatPattern 99
      Visibility <- "System Data_Visible"
      ProcessValue <- "System Data_HMI_Yellow_A"
   IOField "I/O field_2" at 635,320 size 74x24; FormatPattern 99
      Visibility <- "System Data_Visible"
      ProcessValue <- "System Data_HMI_Green_A"
   IOField "I/O field_6" at 634,379 size 74x24; FormatPattern 99
      Visibility <- "System Data_Visible"
      ProcessValue <- "System Data_HMI_Red_A"
   Group "Group" at 209,64 size 41x37
   Group "Group_1" at 155,68 size 43x37
   Button "Button_8" at 711,443 size 86x35; TextOff 'PP1'
      on Click: InvertBit("System Data_Visible")
      on Release: ResetBit("System Data_Enable_PP1")
      on Press: SetBit("System Data_Enable_PP1")
   Button "Button_9" at 627,444 size 84x34; TextOff 'PP2'
      on Click: InvertBit("System Data_Visible_2")
      on Release: ResetBit("System Data_Enalbe_PP2")
      on Press: SetBit("System Data_Enalbe_PP2")
   Button "Button_10" at 544,445 size 84x33; TextOff 'PP3'
      on Release: ResetBit("System Data_Enalbe_PP3")
      on Press: SetBit("System Data_Enalbe_PP3")
   Group "Group_2" at 187,137 size 223x97
   Group "Group_3" at 424,31 size 285x205
   Rectangle "Rectangle_29" at 234,64 size 13x4
      Appearance <- "Data_7SEG_MOD_B"
   Rectangle "Rectangle_30" at 246,68 size 4x14
      Appearance <- "Data_7SEG_MOD_B"
   Rectangle "Rectangle_31" at 234,81 size 13x4
      Appearance <- "Data_7SEG_MOD_B"
   Rectangle "Rectangle_32" at 246,84 size 4x14
      Appearance <- "Data_7SEG_MOD_B"
   Rectangle "Rectangle_33" at 234,97 size 13x4
      Appearance <- "Data_7SEG_MOD_B"
   Rectangle "Rectangle_34" at 231,84 size 4x14
      Appearance <- "Data_7SEG_MOD_B"
   Rectangle "Rectangle_35" at 231,68 size 4x14
      Appearance <- "Data_7SEG_MOD_B"
   Rectangle "Rectangle_1" at 212,64 size 14x4
      Appearance <- "Data_7SEG_DIV_B"
   Rectangle "Rectangle_2" at 225,68 size 4x14
      Appearance <- "Data_7SEG_DIV_B"
   Rectangle "Rectangle_3" at 212,81 size 14x4
      Appearance <- "Data_7SEG_DIV_B"
   Rectangle "Rectangle_4" at 225,84 size 4x14
      Appearance <- "Data_7SEG_DIV_B"
   Rectangle "Rectangle_5" at 212,97 size 14x4
      Appearance <- "Data_7SEG_DIV_B"
   Rectangle "Rectangle_15" at 209,84 size 4x14
      Appearance <- "Data_7SEG_DIV_B"
   Rectangle "Rectangle_21" at 209,68 size 4x14
      Appearance <- "Data_7SEG_DIV_B"
   Rectangle "Rectangle_22" at 181,68 size 14x4
      Appearance <- "Data_7SEG_MOD"
   Rectangle "Rectangle_23" at 194,72 size 4x14
      Appearance <- "Data_7SEG_MOD"
   Rectangle "Rectangle_24" at 181,85 size 14x4
      Appearance <- "Data_7SEG_MOD"
   Rectangle "Rectangle_25" at 194,88 size 4x14
      Appearance <- "Data_7SEG_MOD"
   Rectangle "Rectangle_26" at 181,101 size 14x4
      Appearance <- "Data_7SEG_MOD"
   Rectangle "Rectangle_27" at 178,88 size 4x13
      Appearance <- "Data_7SEG_MOD"
   Rectangle "Rectangle_28" at 178,72 size 4x14
      Appearance <- "Data_7SEG_MOD"
   Rectangle "Rectangle_36" at 158,68 size 14x4
      Appearance <- "Data_7SEG_DIV"
   Rectangle "Rectangle_37" at 171,72 size 4x14
      Appearance <- "Data_7SEG_DIV"
   Rectangle "Rectangle_38" at 158,85 size 14x4
      Appearance <- "Data_7SEG_DIV"
   Rectangle "Rectangle_39" at 171,88 size 4x14
      Appearance <- "Data_7SEG_DIV"
   Rectangle "Rectangle_40" at 158,101 size 14x4
      Appearance <- "Data_7SEG_DIV"
   Rectangle "Rectangle_41" at 155,88 size 4x14
      Appearance <- "Data_7SEG_DIV"
   Rectangle "Rectangle_42" at 155,72 size 4x14
      Appearance <- "Data_7SEG_DIV"
   TextField "Text field_3" at 187,139 size 106x22; Text 'Control Panel'
   Button "Button_1" at 303,138 size 107x32; TextOff '1 Light'
      on Release: ResetBit("System Data_Enable_PP1")
      on Press: SetBit("System Data_Enable_PP1")
      Appearance <- "System Data_Enable_PP1"
      on Click: InvertBit("System Data_Visible")
   Button "Button_3" at 303,170 size 106x32; TextOff '2 Light'
      on Release: ResetBit("System Data_Enalbe_PP2")
      on Press: SetBit("System Data_Enalbe_PP2")
      Appearance <- "System Data_Enalbe_PP2"
      on Click: InvertBit("System Data_Visible_2")
   Button "Button_4" at 303,202 size 106x32; TextOff 'Emergency'
      on Release: ResetBit("System Data_Enalbe_PP3")
      on Press: SetBit("System Data_Enalbe_PP3")
      Appearance <- "System Data_Enalbe_PP3"
   SymbolicIOField "Symbolic I/O field_1" at 187,202 size 118x32; TextOn '1'; TextOff '0'; TextList "Light_mode"
      ProcessValue <- "System Data_Mode"
   Rectangle "Rectangle_7" at 426,31 size 282x205
      Visibility <- "System Data_Visible_2"
   Rectangle "Rectangle_8" at 426,60 size 134x142
      Visibility <- "System Data_Visible_2"
   IOField "I/O field_3" at 488,87 size 67x30; FormatPattern 99
      ProcessValue <- "System Data_HMI_Green_A"
      Visibility <- "System Data_Visible_2"
   IOField "I/O field_4" at 488,123 size 67x30; FormatPattern 99
      ProcessValue <- "System Data_HMI_Yellow_A"
      Visibility <- "System Data_Visible_2"
   IOField "I/O field_5" at 488,160 size 67x30; FormatPattern 99
      ProcessValue <- "Data_Timer_Red A_Value"
      Visibility <- "System Data_Visible_2"
   Button "Button_11" at 635,206 size 73x30; TextOff 'SET'
      on Release: ResetBit("System Data_HMI_SET")
      on Press: SetBit("System Data_HMI_SET")
      Visibility <- "System Data_Visible_2"
   Button "Button_12" at 426,207 size 79x29; TextOff 'Start'
      on Release: ResetBit("System Data_Start")
      on Press: SetBit("System Data_Start")
      Visibility <- "System Data_Visible_2"
   TextField "Text field_9" at 424,56 size 66x26; Text 'Light A'
      Visibility <- "System Data_Visible_2"
   Rectangle "Rectangle_9" at 573,59 size 134x142
      Visibility <- "System Data_Visible_2"
   IOField "I/O field_9" at 635,84 size 67x29; FormatPattern 99
      ProcessValue <- "System Data_HMI_Green_B"
      Visibility <- "System Data_Visible_2"
   IOField "I/O field_10" at 635,122 size 67x29; FormatPattern 99
      ProcessValue <- "System Data_HMI_Yellow_B"
      Visibility <- "System Data_Visible_2"
   IOField "I/O field_11" at 635,159 size 67x29; FormatPattern 99
      ProcessValue <- "Data_Timer_Red B_Value"
      Visibility <- "System Data_Visible_2"
   TextField "Text field_10" at 572,54 size 66x29; Text 'Light B'
      Visibility <- "System Data_Visible_2"
   TextField "Text field_4" at 429,92 size 56x27; Text 'Green'
      Visibility <- "System Data_Visible_2"
   TextField "Text field_5" at 431,123 size 56x27; Text 'Yellow'
      Visibility <- "System Data_Visible_2"
   TextField "Text field_13" at 428,159 size 56x27; Text 'Red'
      Visibility <- "System Data_Visible_2"
   TextField "Text field_14" at 576,86 size 56x26; Text 'Green'
      Visibility <- "System Data_Visible_2"
   TextField "Text field_15" at 579,122 size 56x26; Text 'Yellow'
      Visibility <- "System Data_Visible_2"
   TextField "Text field_16" at 573,158 size 56x26; Text 'Red'
      Visibility <- "System Data_Visible_2"
   Button "Button_14" at 631,32 size 78x27; TextOff 'X'
      on Click: InvertBit("System Data_Visible_2")
      Visibility <- "System Data_Visible_2"
   Button "Button_15" at 504,207 size 78x29; TextOff 'Stop'
      on Release: ResetBit("System Data_Stop")
      on Press: SetBit("System Data_Stop")
      Appearance <- "System Data_Stop"
      Visibility <- "System Data_Visible_2"
*)

(* ===== HMI "HMI_RT_2" =====
system functions are stored by id; their names below are inferred from use
connection "HMI_Connection_9": ETHERNET, S7_1500_OMS

HMI tags "Default tag table"
   "System Data_Green A" : Bool = PLC "System Data"."Green A" AT %DB1.DBX0.0, 1 s
   "System Data_Yellow A" : Bool = PLC "System Data"."Yellow A" AT %DB1.DBX0.0, 1 s
   "System Data_Red A" : Bool = PLC "System Data"."Red A" AT %DB1.DBX0.0, 1 s
   "System Data_Green B" : Bool = PLC "System Data"."Green B" AT %DB1.DBX0.0, 1 s
   "System Data_Yellow B" : Bool = PLC "System Data"."Yellow B" AT %DB1.DBX0.0, 1 s
   "System Data_Red B" : Bool = PLC "System Data"."Red B" AT %DB1.DBX0.0, 1 s
   "System Data_Start" : Bool = PLC "System Data".Start AT %DB1.DBX0.0, 1 s
   "Timer1_ET" : Time = PLC Timer1.ET AT %DB1.DBD0, 1 s
   "Timer2_ET" : Time = PLC Timer2.ET AT %DB1.DBD0, 1 s
   "Timer3_ET" : Time = PLC Timer3.ET AT %DB1.DBD0, 1 s
   "Timer4_Q" : Bool = PLC Timer4.Q AT %DB1.DBX0.0, 1 s
   "Timer4_ET" : Time = PLC Timer4.ET AT %DB1.DBD0, 1 s
   "System Data_Green A _Value" : DInt = PLC "System Data"."Green A _Value" AT %DB1.DBD0, 1 s
   "System Data_Green B_Value" : DInt = PLC "System Data"."Green B_Value" AT %DB1.DBD0, 1 s
   "System Data_HMI_SET" : Bool = PLC "System Data".HMI_SET AT %DB1.DBX0.0, 1 s
   "System Data_HMI_Green_A" : DInt = PLC "System Data".HMI_Green_A AT %DB1.DBD0, 1 s
   "System Data_HMI_Green_B" : DInt = PLC "System Data".HMI_Green_B AT %DB1.DBD0, 1 s
   "System Data_Stop" : Bool = PLC "System Data".Stop AT %DB1.DBX0.0, 1 s
   "T1_ET" : Time = PLC T1.ET AT %DB1.DBD0, 1 s
   "System Data_Enable_PP1" : Bool = PLC "System Data".Enable_PP1 AT %DB1.DBX0.0, 1 s
   "System Data_Enalbe_PP2" : Bool = PLC "System Data".Enalbe_PP2 AT %DB1.DBX0.0, 1 s
   "System Data_Cancel" : Bool = PLC "System Data".Reset AT %DB1.DBX0.0, 1 s
   "System Data_Enalbe_PP3" : Bool = PLC "System Data".Enalbe_PP3 AT %DB1.DBX0.0, 1 s
   "System Data_HMI_Yellow_A" : DInt = PLC "System Data".HMI_Yellow_A AT %DB1.DBD0, 1 s
   "System Data_HMI_Yellow_B" : DInt = PLC "System Data".HMI_Yellow_B AT %DB1.DBD0, 1 s
   "Data_Timer_Red A_Value" : DInt = PLC Data."Red A_Value" AT %DB1.DBD0, 1 s
   "Data_Timer_Red B_Value" : DInt = PLC Data."Red B_Value" AT %DB1.DBD0, 1 s
   "Data_7SEG_DIV" : Byte = PLC Data.7SEG_DIV_A AT %DB1.DBB0, 1 s
   "Data_7SEG_MOD" : Byte = PLC Data.7SEG_MOD_A AT %DB1.DBB0, 1 s
   "Data_7SEG_DIV_B" : Byte = PLC Data.7SEG_DIV_B AT %DB1.DBB0, 1 s
   "Data_7SEG_MOD_B" : Byte = PLC Data.7SEG_MOD_B AT %DB1.DBB0, 1 s
   "System Data_HMI_Red_A" : DInt = PLC "System Data".HMI_Red_A AT %DB1.DBD0, 1 s
   "System Data_HMI_Red_B" : DInt = PLC "System Data".HMI_Red_B AT %DB1.DBD0, 1 s
   "Data_TIme_LIGHT_A" : DInt = PLC Data.TIme_LIGHT_A, 1 s
   "Data_Time_LIGHT_B" : DInt = PLC Data.Time_LIGHT_B, 1 s
   "Data_Remain_DEC_A" : Int = PLC Data.Remain_DEC_A, 1 s
   "Data_Remain_DEC_B" : Int = PLC Data.Remain_DEC_B, 1 s
   "System Data_Visible" : Bool = PLC "System Data".Visible_1, 1 s
   "System Data_Mode" : DInt = PLC "System Data".Mode, 1 s

text list "Light_mode": 1 '1 Light'; 2 '2 Light'; 3 'Emergency'; 0 'Stop'

screen "Screen_1" 1024x768
   TextField "Text field_1" at 183,10 size 345x44; Text 'TRAFFIC LIGHT CONTROL'
   Group "Group" at 30,131 size 223x97
   TextField "Text field_3" at 21,51 size 337x80; Text 'Student: Võ Quang Thanh Nghĩa ID: 1851093'
   TextField "Text field_2" at 30,133 size 106x22; Text 'Control Panel'
   Button "Button_2" at 146,132 size 107x32; TextOff '1 Light'
      on Press: SetBit("System Data_Enable_PP1")
      on Release: ResetBit("System Data_Enable_PP1")
      Appearance <- "System Data_Enable_PP1"
      on Click: function_efd93a16("Option1", 400, 100, -1, -1, 1)
   Button "Button_5" at 146,164 size 106x32; TextOff '2 Light'
      on Press: SetBit("System Data_Enalbe_PP2")
      on Release: ResetBit("System Data_Enalbe_PP2")
      Appearance <- "System Data_Enalbe_PP2"
      on Click: function_efd93a16("Option2", 400, 100, -1, -1, 1)
   Button "Button_7" at 146,196 size 106x32; TextOff 'Emergency'
      on Press: SetBit("System Data_Enalbe_PP3")
      on Release: ResetBit("System Data_Enalbe_PP3")
      Appearance <- "System Data_Enalbe_PP3"
   SymbolicIOField "Symbolic I/O field_1" at 30,196 size 118x32; TextOff '0'; TextOn '1'; TextList "Light_mode"
      ProcessValue <- "System Data_Mode"

PopupScreen "Option1" 350x318
   Button "Button_3" at 272,276 size 76x38; TextOff 'SET'
      on Release: ResetBit("System Data_HMI_SET")
      on Press: SetBit("System Data_HMI_SET")
   Button "Button_1" at 105,276 size 86x38; TextOff 'Start'
      on Release: ResetBit("System Data_Start")
      on Press: SetBit("System Data_Start")
   Button "Button_4" at 191,276 size 81x38; TextOff 'Stop'
      on Release: ResetBit("System Data_Stop")
      on Press: SetBit("System Data_Stop")
   Button "Button_5" at 258,1 size 91x35; TextOff 'X'
      on Click: function_efd93a16("Option1", 0, 0, 0, -1, 1)
   Group "Group_2" at 8,4 size 90x82
   TextField "Text field_3" at 116,85 size 69x29; Text 'LIGHT'
   TextField "Text field_5" at 113,118 size 69x30; Text 'Green'
   TextField "Text field_6" at 113,165 size 69x30; Text 'Yellow'
   TextField "Text field_7" at 114,205 size 69x30; Text 'Red'
   IOField "I/O field_4" at 184,161 size 87x36; FormatPattern 99
      ProcessValue <- "System Data_HMI_Yellow_A"
   IOField "I/O field_3" at 184,116 size 87x36; FormatPattern 99
      ProcessValue <- "System Data_HMI_Green_A"
   IOField "I/O field_5" at 184,205 size 87x36; FormatPattern 99
      ProcessValue <- "System Data_HMI_Red_A"
   IOField "I/O field_7" at 115,48 size 100x36; FormatPattern 99
      ProcessValue <- "Data_Remain_DEC_A"
   Group "Group" at 0,88 size 108x224
   Circle "Circle_1" at 24,98 size 55x55
      Appearance <- "System Data_Green A"
   Circle "Circle_2" at 24,170 size 55x55
      Appearance <- "System Data_Yellow A"
   Circle "Circle_3" at 24,242 size 55x55
      Appearance <- "System Data_Red A"
   Rectangle "Rectangle_7" at 42,10 size 8x34
      Appearance <- "Data_7SEG_DIV"
   Rectangle "Rectangle_6" at 16,4 size 27x7
      Appearance <- "Data_7SEG_DIV"
   Rectangle "Rectangle_8" at 16,43 size 27x7
      Appearance <- "Data_7SEG_DIV"
   Rectangle "Rectangle_9" at 43,49 size 8x30
      Appearance <- "Data_7SEG_DIV"
   Rectangle "Rectangle_10" at 15,78 size 29x8
      Appearance <- "Data_7SEG_DIV"
   Rectangle "Rectangle_11" at 9,49 size 8x30
      Appearance <- "Data_7SEG_DIV"
   Rectangle "Rectangle_12" at 8,10 size 8x33
      Appearance <- "Data_7SEG_DIV"
   Rectangle "Rectangle_13" at 64,5 size 26x8
      Appearance <- "Data_7SEG_MOD"
   Rectangle "Rectangle_14" at 89,12 size 8x32
      Appearance <- "Data_7SEG_MOD"
   Rectangle "Rectangle_16" at 64,43 size 26x7
      Appearance <- "Data_7SEG_MOD"
   Rectangle "Rectangle_17" at 90,50 size 8x29
      Appearance <- "Data_7SEG_MOD"
   Rectangle "Rectangle_18" at 64,78 size 27x8
      Appearance <- "Data_7SEG_MOD"
   Rectangle "Rectangle_19" at 57,48 size 8x31
      Appearance <- "Data_7SEG_MOD"
   Rectangle "Rectangle_20" at 57,12 size 8x32
      Appearance <- "Data_7SEG_MOD"

PopupScreen "Option2" 561x349
   IOField "I/O field_8" at 109,312 size 98x33; FormatPattern 99
      ProcessValue <- "Data_Remain_DEC_B"
   IOField "I/O field_7" at 2,313 size 98x32; FormatPattern 99
      ProcessValue <- "Data_Remain_DEC_A"
   Circle "Circle_1" at 24,97 size 48x48
      Appearance <- "System Data_Green A"
   Circle "Circle_2" at 24,170 size 48x48
      Appearance <- "System Data_Yellow A"
   Circle "Circle_3" at 24,243 size 48x48
      Appearance <- "System Data_Red A"
   Circle "Circle_4" at 134,98 size 48x48
      Appearance <- "System Data_Green B"
   Circle "Circle_5" at 132,169 size 48x48
      Appearance <- "System Data_Yellow B"
   Circle "Circle_6" at 131,242 size 48x48
      Appearance <- "System Data_Red B"
   Group "Group_1" at 6,4 size 90x82
   Group "Group_2" at 107,5 size 95x80
   IOField "I/O field_3" at 293,145 size 76x33; FormatPattern 99
      ProcessValue <- "System Data_HMI_Green_A"
   IOField "I/O field_4" at 293,185 size 76x33; FormatPattern 99
      ProcessValue <- "System Data_HMI_Yellow_A"
   IOField "I/O field_5" at 293,226 size 76x33; FormatPattern 99
      ProcessValue <- "Data_Timer_Red A_Value"
   Button "Button_3" at 475,291 size 82x32; TextOff 'SET'
      on Release: ResetBit("System Data_HMI_SET")
      on Press: SetBit("System Data_HMI_SET")
   Button "Button_1" at 214,290 size 89x32; TextOff 'Start'
      on Release: ResetBit("System Data_Start")
      on Press: SetBit("System Data_Start")
   Button "Button_4" at 303,290 size 91x32; TextOff 'Stop'
      on Release: ResetBit("System Data_Stop")
      on Press: SetBit("System Data_Stop")
   TextField "Text field_3" at 221,110 size 74x29; Text 'Light A'
   IOField "I/O field_9" at 459,145 size 76x32; FormatPattern 99
      ProcessValue <- "System Data_HMI_Green_B"
   IOField "I/O field_10" at 459,185 size 76x32; FormatPattern 99
      ProcessValue <- "System Data_HMI_Yellow_B"
   IOField "I/O field_11" at 459,226 size 76x32; FormatPattern 99
      ProcessValue <- "Data_Timer_Red B_Value"
   TextField "Text field_4" at 388,109 size 75x32; Text 'Light B'
   TextField "Text field_5" at 226,150 size 63x30; Text 'Green'
   TextField "Text field_6" at 229,185 size 63x30; Text 'Yellow'
   TextField "Text field_7" at 225,225 size 63x30; Text 'Red'
   TextField "Text field_8" at 392,145 size 63x29; Text 'Green'
   TextField "Text field_9" at 396,185 size 63x29; Text 'Yellow'
   TextField "Text field_10" at 389,225 size 63x29; Text 'Red'
   Button "Button_5" at 474,0 size 86x35; TextOff 'X'
      on Click: function_efd93a16("Option2", 0, 0, 0, -1, 1)
   Rectangle "Rectangle_6" at 14,4 size 27x7
      Appearance <- "Data_7SEG_DIV"
   Rectangle "Rectangle_7" at 40,10 size 8x34
      Appearance <- "Data_7SEG_DIV"
   Rectangle "Rectangle_8" at 14,43 size 27x7
      Appearance <- "Data_7SEG_DIV"
   Rectangle "Rectangle_9" at 41,49 size 8x30
      Appearance <- "Data_7SEG_DIV"
   Rectangle "Rectangle_10" at 13,78 size 29x8
      Appearance <- "Data_7SEG_DIV"
   Rectangle "Rectangle_11" at 7,49 size 8x30
      Appearance <- "Data_7SEG_DIV"
   Rectangle "Rectangle_12" at 6,10 size 8x33
      Appearance <- "Data_7SEG_DIV"
   Rectangle "Rectangle_13" at 62,5 size 26x8
      Appearance <- "Data_7SEG_MOD"
   Rectangle "Rectangle_14" at 87,12 size 8x32
      Appearance <- "Data_7SEG_MOD"
   Rectangle "Rectangle_16" at 62,43 size 26x7
      Appearance <- "Data_7SEG_MOD"
   Rectangle "Rectangle_17" at 88,50 size 8x29
      Appearance <- "Data_7SEG_MOD"
   Rectangle "Rectangle_18" at 62,78 size 27x8
      Appearance <- "Data_7SEG_MOD"
   Rectangle "Rectangle_19" at 55,48 size 8x31
      Appearance <- "Data_7SEG_MOD"
   Rectangle "Rectangle_20" at 55,12 size 8x32
      Appearance <- "Data_7SEG_MOD"
   Rectangle "Rectangle_22" at 114,5 size 26x8
      Appearance <- "Data_7SEG_DIV_B"
   Rectangle "Rectangle_23" at 139,13 size 8x32
      Appearance <- "Data_7SEG_DIV_B"
   Rectangle "Rectangle_24" at 114,44 size 26x7
      Appearance <- "Data_7SEG_DIV_B"
   Rectangle "Rectangle_25" at 139,50 size 8x29
      Appearance <- "Data_7SEG_DIV_B"
   Rectangle "Rectangle_26" at 115,78 size 25x7
      Appearance <- "Data_7SEG_DIV_B"
   Rectangle "Rectangle_27" at 107,51 size 8x28
      Appearance <- "Data_7SEG_DIV_B"
   Rectangle "Rectangle_28" at 107,12 size 8x32
      Appearance <- "Data_7SEG_DIV_B"
   Rectangle "Rectangle_29" at 168,5 size 26x8
      Appearance <- "Data_7SEG_MOD_B"
   Rectangle "Rectangle_30" at 193,13 size 8x32
      Appearance <- "Data_7SEG_MOD_B"
   Rectangle "Rectangle_31" at 168,44 size 27x7
      Appearance <- "Data_7SEG_MOD_B"
   Rectangle "Rectangle_32" at 194,50 size 8x28
      Appearance <- "Data_7SEG_MOD_B"
   Rectangle "Rectangle_33" at 168,77 size 27x8
      Appearance <- "Data_7SEG_MOD_B"
   Rectangle "Rectangle_34" at 161,50 size 8x28
      Appearance <- "Data_7SEG_MOD_B"
   Rectangle "Rectangle_35" at 161,13 size 8x32
      Appearance <- "Data_7SEG_MOD_B"

